# B&R Automation Studio project 305841_E00002_0 (part 10)

#### AxSMInit.st
```iecst
PROGRAM _INIT
  // set ax pointer to the element of the global sMot_Axis array
  ax ACCESS ADR(axes[AXIS_NO]);

  // set the position limits to point to the global permanent variable
  axPositionLimits ACCESS ADR(gr_AxisPositionLimits[AXIS_NO]);

  // Set the axis number and clear the ignore bit
  ax.AxisNo:= AXIS_NO;

  // **** These settings need to be reviewed/set for each axis
  ax.CouplingParameters.SlaveAxisNo := DINT_TO_USINT(AD_UNKNOWN); // No slaves for the CF VFD
  ax.Ignore := FALSE;
  ax.isAxisEndless := TRUE;
  ax.isAxisVirtual := FALSE;
  ax.isAxisInverter := TRUE;

  // Point to the mappMotion axis, and a slave if there is one
  ax.AxisObj := gAxCfPmp; // mappMotion axis -- see mappMotion in cfg view
  ax.SlaveAxisObj := axDummySlave; // slave axis for the handwheel is dynamic

  // Set the restore pos check fb
  // ax.fbCheckRestorePos.Axis := ADR(ax.AxisObj);
  // ax.fbCheckRestorePos.DataAddress := ADR(gr_AxCfVfdRestorePos); // Set this per axis

  // Load the min/max velocity and accel/decel from constants
  ax.MoveParameters.AccelMin := 0.001; // TODO: Not sure of a good value, but it should not be zero.
  ax.MoveParameters.AccelMax := AXIS_CFVFD_MAX_ACCEL;
  ax.MoveParameters.DecelMin := 0.001; // TODO:Not sure of a good value, but it should not be zero.
  ax.MoveParameters.DecelMax:= AXIS_CFVFD_MAX_DECEL;
  ax.MoveParameters.VelocityMin := 0.000;
  ax.MoveParameters.VelocityMax := AXIS_CFVFD_MAX_VELOCITY;

  // **** The settings below don't normally need to be altered

  // set the fb axis references
  ax.fbMpAxisBasic.MpLink := ADR(ax.AxisObj);
  ax.fbReadDrivePos.Axis:= ADR(ax.AxisObj);
  ax.fbGearIn.Master := ADR(ax.AxisObj);
  ax.fbGearIn.Slave := ADR(ax.SlaveAxisObj);
  ax.fbGearOut.Slave := ADR(ax.SlaveAxisObj);
  ax.fbOffsetShift.Slave := ADR(ax.SlaveAxisObj);
  ax.fbPhaseShift.Slave := ADR(ax.SlaveAxisObj);
  ax.fbCamIn.Master := ADR(ax.AxisObj);
  ax.fbCamIn.Slave := ADR(ax.SlaveAxisObj);
  ax.fbCamOut.Slave := ADR(ax.SlaveAxisObj);
  ax.fbUpdateBFbParams._I_Axis := ADR(ax);

  // Set fb reference to local variables
  ax.fbMpAxisBasic.Parameters := ADR(axisBasicParams);

  // Set previous values for motion parameters so changes can be detected
  ax.MoveParametersPrev := ax.MoveParameters;

  // Clear commands and requests
  fctClearMotionCommands(_I_CmdMask := MACM_NOMASK, _IO_Commands := ax.Commands);
  fctClearMotionRequests(_I_ReqMask := MACM_NOMASK, _IO_Commands := ax.Commands);

  // set the move not allowed flag
  ax.Commands.MoveNotAllowed:= TRUE;

  // Set the most primitive status. If the axis is valid, the
  // full status will be updated later once comms is established, and the drive status is updated via MpAxisBasic
  ax.Status.IsCommuncationReady := FALSE;
  ax.Status.IsReadyToPowerOn := FALSE;

END_PROGRAM
```

### Program Logical/PlcLogic/CutProfile/CutProfileCam (IEC) - Calcs and function calls needed to turn the cut profile into a loaded CAM table.

#### CutProfileCam.var - Local variables
```iecst
VAR CONSTANT
  CAM_POINTS : UINT := 250;
END_VAR

VAR

  (* program control *)
  seqCtr : SINT; (* sequence counter *)
  idx : UINT; (* index *)

  (****** Cam related ******)
  (* program control for cam creation *)
  reqCreateCamTable : BOOL := FALSE; (* request to start seq *)
  createCamTableOS : BOOL := FALSE;
  createCamTableDone : BOOL := FALSE;
  camTableId : UINT := 14; (* 1-14, but data type compatible with cam prepare fb *)
  camSeqCtr : SINT; (* sequence counter *)
  camTable : McCamSectionsType; (* local cam sections table *)
  camData : McCamDataType; (* cam data calculated from sections *)
  camPointsMaster : ARRAY[0..CAM_POINTS] OF LREAL;
  camPointsSlave : ARRAY[0..CAM_POINTS] OF LREAL;
  fbCreateCamSections : fbCalcCamSections;
  fbCalcCamFromSections : MC_BR_CalcCamFromSections;
  fbCalcCamPoints : MC_BR_CalcPointsFromCam;
  fbCamPrepare : MC_BR_CamPrepare;
  (* detect changes to cut profile *)
  cutProfileCamLoadedPrev : sWp_CuttingHead; (* previous cut profile loaded into the cam table. *)
  (* BR Str mem fct params *)
  cutProfileBytes : UDINT;
  result : DINT;
  nxtAddr : UDINT;

  (****** Recipe and file related ******)

  (* Local version of the lookup table *)
	depthToAngleLu : sXYTableLu150;

  (* program control for directory creation *)
  reqInitDirs : BOOL := FALSE; (* request to start seq *)
  initDirsOS : BOOL := FALSE;
  initDirsDone : BOOL := FALSE;
  devName : STRING[80]; (* also used for recipe read *)
  dirName : STRING[255];

  (* program control for Depth To Angle Lu recipe registration *)
  pvNameLocalDepthToAngleLu : STRING[100];
  pvNameGloballDepthToAngleLu : STRING[100];
  pvCatagoryDepthToAngleLu : STRING[50];

  (* program control for recipe read/write *)
  recipeReadOverwiteGlobal : BOOL := FALSE;

  recipeReadFileName : STRING[255];
  recipeWriteFileName : STRING[255];

  reqRecipeReadAngleLu : BOOL := FALSE;
  recipeReadAngleLuOS : BOOL := FALSE;
  recipeReadAngleLuDone : BOOL := FALSE;

  reqRecipeWriteAngleLu : BOOL := FALSE;
  recipeWriteAngleLuOS : BOOL := FALSE;
  recipeWriteAngleLuDone : BOOL := FALSE;
  csvHeader : MpRecipeCsvHeaderType;

  (* FileIO fbs *)
  fbDirCreate : DirCreate;

  (* recipe fbs *)
  fbRcpiRegLocalDToALu : MpRecipeRegPar; (* register local Depth To Angle Lu Table to recipe *)
  fbRcpiRegGlobalDToALu : MpRecipeRegPar; (* register global Depth To Angle Lu Table to recipe *)
  fbRecipeCsv : MpRecipeCsv; (* recipe to/from file *)

END_VAR
```

#### CutProfileCam.st - Cyclic code
```iecst
PROGRAM _INIT

  (****** Cam related ******)
  // Set up fb to populate cam sections
  fbCreateCamSections.CamTable := ADR(camTable);
  fbCreateCamSections.DepthToAngle_T1 := ADR(gr_depthToAngleLu.T1);
  fbCreateCamSections.DepthToAngle_T2 := ADR(gr_depthToAngleLu.T2);
  fbCreateCamSections.DepthToAngle_T3 := ADR(gr_depthToAngleLu.T3);
  // Get the length of the cut profile parts of the cutting head configuration
  // This aids in change detection
  cutProfileBytes := ADR(gr_CfgCurrent.cuttingHead.EndOfCutProfile) - ADR(gr_CfgCurrent.cuttingHead.StartOfCutProfile);

  (****** Recipe and file related ******)

  // Setup registration of PV to a recipe
  // Each PV uses a separate registration FB
  // Local Depth To Angle LU Table
  // Use local LU table for recipe access and transfer to/from global when all is well
  pvNameLocalDepthToAngleLu := 'CrCamTbl:depthToAngleLu';
  pvCatagoryDepthToAngleLu := 'DepthToAngle';
  fbRcpiRegLocalDToALu.MpLink := ADR(angleLuRecipeCsv);
  fbRcpiRegLocalDToALu.Enable := FALSE;
  fbRcpiRegLocalDToALu.ErrorReset := FALSE;
  fbRcpiRegLocalDToALu.PVName := ADR(pvNameLocalDepthToAngleLu);
  fbRcpiRegLocalDToALu.Category := ADR(pvCatagoryDepthToAngleLu);
  // set up the fb by calling with enable false, and then set enable
  // true so it is ready to go in cyclic.
  fbRcpiRegLocalDToALu();
  fbRcpiRegLocalDToALu.Enable := TRUE;

  // Global Depth To Angle LU Table
  // Use local LU table for recipe access and transfer to/from global when all is well
  pvNameGloballDepthToAngleLu := 'gr_depthToAngleLu';
  pvCatagoryDepthToAngleLu := 'DepthToAngle';
  fbRcpiRegGlobalDToALu.MpLink := ADR(angleLuRecipeCsv);
  fbRcpiRegGlobalDToALu.Enable := FALSE;
  fbRcpiRegGlobalDToALu.ErrorReset := FALSE;
  fbRcpiRegGlobalDToALu.PVName := ADR(pvNameGloballDepthToAngleLu);
  fbRcpiRegGlobalDToALu.Category := ADR(pvCatagoryDepthToAngleLu);
  // set up the fb by calling with enable false, and then set enable
  // true so it is ready to go in cyclic.
  fbRcpiRegGlobalDToALu();
  fbRcpiRegGlobalDToALu.Enable := TRUE;

  // Set flag to create directories
  reqInitDirs := TRUE; // true will trigger dir setup (creation) after startup
  initDirsOS := FALSE;
  initDirsDone := FALSE;

  // Set flags to control read/write of recipes
  // recipe file names
  recipeReadFileName := 'DepthToAngleLookup_recipe_b.csv';
  recipeWriteFileName := 'DepthToAngleLookup_recipe_b_FromPlc.csv';

  // set whether or not to overwrite the global data on sucessful local read
  recipeReadOverwiteGlobal := FALSE;

  reqRecipeReadAngleLu := FALSE; // set high to read recipe after startup
  recipeReadAngleLuOS := FALSE;
  recipeReadAngleLuDone := FALSE;

  reqRecipeWriteAngleLu := FALSE; // set high to write recipe after startup
  recipeWriteAngleLuOS := FALSE;
  recipeWriteAngleLuDone := FALSE;

 END_PROGRAM

PROGRAM _CYCLIC

  // *****************
  // Cam table: Detect cut profile changes
  // *****************
  // result = brsmemcmp(ADR(Mem1),ADR(Mem2),length), result = 0 when equal
  result := brsmemcmp(ADR(cutProfileCamLoadedPrev.StartOfCutProfile),
                      ADR(gr_CfgCurrent.cuttingHead.StartOfCutProfile),
                      cutProfileBytes);
  // Enable loading the CAM table if it has not been done yet,
  // or if a change is detected, or if the last time there was an error,
  // but the machine cannot be in cycle while a cam table change in made.
  hmiProcessReqs.calCalcTableEnable := (result <> 0 OR NOT createCamTableDone OR camSeqCtr < -1);
  // If a change has been detected, but the table has not been sucessfully loaded, clear the part motion flag
  IF  hmiProcessReqs.calCalcTableEnable AND createCamTableOS THEN
    partMotion.camTableLoaded := FALSE;
  END_IF;

  // *****************
  // Create Cam table on request
  // *****************
  // Set the create cam table request and clear the HMI request upon an HMI request.
  // The logic will handle the rest.
  IF hmiProcessReqs.camReqCalcTable THEN
    reqCreateCamTable := TRUE;
    hmiProcessReqs.camReqCalcTable := FALSE;
  END_IF;

  // On request, calculate and populate cam sections base on cut parameters.
  // Done sucessfully, and camSeqCtr should start from 1, go up, and then end up at -1.
  // Errors result in a more negative camSeqCtr
  // TODO: Deal with errors. Right now the sequence stops, with the camSeqCtr being set to
  // a value more negative than -1.

  IF reqCreateCamTable THEN

    // if the OS is clear, this is the first time thru ...
    // init the seq number and manage flags and OS
    IF NOT createCamTableOS THEN
      // Set the OS so this bit only happens once per req
      createCamTableOS := TRUE;
      // Init the seq ctr
      camSeqCtr := 1;
      // Clear the done flag
      createCamTableDone := FALSE;
      // Clear the hmi request
      hmiProcessReqs.camReqCalcTable := FALSE;
    END_IF;

    IF 1 = camSeqCtr THEN
      // Use cam id 14 for calculated cam table
      camTableId := PROD_CAM_TABLE_ID;
      // Guess the operator will use this cam id
      // TODO: No access to hmiLibraryAxisReqs in OmSaveDev!!

      // Set up to calc the cam sections fb
      // Use the current cutting head configuration for the cut profile

      // Force the finish pass depth to be zero if the option is not chosen
      IF gr_CfgCurrent.cuttingHead.finishingPass THEN
        fbCreateCamSections.FinishPassDepth :=  gr_CfgCurrent.cuttingHead.finishingPassDepth;
      ELSE
        fbCreateCamSections.FinishPassDepth := 0.0;
      END_IF;
      fbCreateCamSections.PassCount := gr_CfgCurrent.cuttingHead.passCount;
      fbCreateCamSections.FinalDepth := gr_CfgCurrent.cuttingHead.totalDepth;
      fbCreateCamSections.CutInAngle := LREAL_TO_REAL(gr_CfgCurrent.cuttingHead.depthAdjAngle);
      fbCreateCamSections.OverCutAngle := LREAL_TO_REAL(gr_CfgCurrent.cuttingHead.cutOverrunAngle);

      // Clear the camTable, camData, and point arrays
      // nxt_adr := brsmemset(ADR(Mem),value,length);
      nxtAddr := brsmemset(ADR(camTable), 0, SIZEOF(camTable));
      nxtAddr := brsmemset(ADR(camData), 0, SIZEOF(camData));
      nxtAddr := brsmemset(ADR(camPointsMaster), 0, SIZEOF(camPointsMaster));
      nxtAddr := brsmemset(ADR(camPointsSlave), 0, SIZEOF(camPointsSlave));

      // Call with enable false to make sure everything is reset and ready to execute with new info
      fbCreateCamSections.Enable := FALSE;
      fbCreateCamSections();
      // onto the next step
      camSeqCtr := 2;
    ELSIF 2 = camSeqCtr THEN
      // Calc the cam sections
      fbCreateCamSections.Enable := TRUE;
      fbCreateCamSections();
      IF fbCreateCamSections.Done AND NOT fbCreateCamSections.Error THEN
        // All done and no error. Move on ...
        // Reset FB and go to next step
        fbCreateCamSections.Enable := FALSE;
        fbCreateCamSections();
        camSeqCtr := 3;
      ELSIF fbCreateCamSections.Done AND fbCreateCamSections.Error THEN
        // Done with an error. Bail out ...
        camSeqCtr := -2;
      END_IF;
    ELSIF 3 = camSeqCtr THEN
      // Set up to calc the cam from the sections
      fbCalcCamFromSections.CamSectionsAddress := ADR(camTable);
      fbCalcCamFromSections.CamDataAddress := ADR(camData);
      // Call with execute false to make sure everything is reset and ready to execute with new info
      fbCalcCamFromSections.Execute := FALSE;
      fbCalcCamFromSections();
      // onto the next step
      camSeqCtr := 4;
    ELSIF 4 = camSeqCtr THEN
      // Calc the cam sections
      fbCalcCamFromSections.Execute := TRUE;
      fbCalcCamFromSections();
      IF fbCalcCamFromSections.Done AND NOT fbCalcCamFromSections.Error THEN
        // All done and no error. Move on ...
        // Reset FB and go to next step
        fbCalcCamFromSections.Execute := FALSE;
        fbCalcCamFromSections();
        camSeqCtr := 5;
      ELSIF NOT fbCalcCamFromSections.Busy AND fbCalcCamFromSections.Error THEN
        // Done with an error. Bail out ...
        camSeqCtr := -4;
      END_IF;
    ELSIF 5 = camSeqCtr THEN
      // Set up to prepare and load the cam data
      fbCamPrepare.Axis := ADR(axes[AD_INNER_ECCENTRIC].AxisObj);
      fbCamPrepare.Cam.DataObjectName := ''; // not used if Cam.DataAdress <> 0
      fbCamPrepare.Cam.DataAdress := ADR(camData); // cam data calculated in fbCalcCamFromSections
      fbCamPrepare.CamID := camTableId;
      // Call with execute false to make sure everything is reset and ready to execute with new info
      fbCamPrepare.Execute := FALSE;
      fbCamPrepare();
      // onto the next step
      camSeqCtr := 6;
    ELSIF 6 = camSeqCtr THEN
      // Prepare and load the cam data
      fbCamPrepare.Execute := TRUE;
      fbCamPrepare();
      IF fbCamPrepare.Done AND NOT fbCamPrepare.Error THEN
        // All done and no error. Move on ...
        // Reset FB and go to next step
        fbCamPrepare.Execute := FALSE;
        fbCamPrepare();
        camSeqCtr := -1;  // TEST: skip fbCalcCamPoints. Getting an error
      ELSIF NOT fbCamPrepare.Busy AND fbCamPrepare.Error THEN
        // Done with an error. Bail out ...
        camSeqCtr := -6;
      END_IF;
    ELSIF 7 = camSeqCtr THEN
      // Set up to calculate cam points
      fbCalcCamPoints.Cam.DataObjectName := ''; // not used if Cam.DataAdress <> 0
      fbCalcCamPoints.Cam.DataAdress := ADR(camData); // cam data calculated in fbCalcCamFromSections
      fbCalcCamPoints.MasterPointsAddress := ADR(camPointsMaster);
      fbCalcCamPoints.SlavePointsAddress := ADR(camPointsSlave);
      fbCalcCamPoints.NumberOfPoints := CAM_POINTS;
      // Call with execute false to make sure everything is reset and ready to execute with new info
      fbCalcCamPoints.Execute := FALSE;
      fbCalcCamPoints();
      // onto the next step
      camSeqCtr := 8;
    ELSIF 8 = camSeqCtr THEN
      // Calcuate points from the cam data
      fbCalcCamPoints.Execute := TRUE;
      fbCalcCamPoints();
      IF fbCalcCamPoints.Done AND NOT fbCalcCamPoints.Error THEN
        // All done and no error. Move on ...
        // reset fb
        fbCalcCamPoints.Execute := FALSE;
        fbCalcCamPoints();
        camSeqCtr := -1;
      ELSIF NOT fbCalcCamPoints.Busy AND fbCalcCamPoints.Error THEN
        // Done with an error. Bail out ...
        camSeqCtr := -8;
      END_IF;
    ELSIF -1 = camSeqCtr THEN
      // All done making cam sections.
      // Getting ready if another request is made.
      // Clear the createCamTable flag and OS and set the done.
      reqCreateCamTable := FALSE;
      createCamTableOS := FALSE; // clear the OS so another initDirs resets things up top
      createCamTableDone := TRUE;
      // Set the flag in part motion
      partMotion.camTableLoaded := TRUE;
      // reset fb
      fbCreateCamSections.Enable := FALSE;
      fbCreateCamSections();
      // Update the previous cut profile values so changes can be detected
      // nxtAddr = brsmemcpy(adr(Dest),adr(Src),length)
      nxtAddr := brsmemcpy(ADR(cutProfileCamLoadedPrev.StartOfCutProfile),
                           ADR(gr_CfgCurrent.cuttingHead.StartOfCutProfile),
                           cutProfileBytes);
    END_IF;
  ELSE
    // createCamTable is false. Clear the OS so we can one time thru it next time
    createCamTableOS := FALSE;
  END_IF;

  // *****************
  // Set up directories
  // *****************
  // Execute FileIO DirCreate async until done or error
  // seqCtr odd: set up DirCreate fb
  // seqCtr even : create dir
  // Use the OS so the directory management can be easily re-run
  // by setting initDirs true (again)
  IF reqInitDirs THEN
    // if the OS is clear, this is the first time thru ...
    // init the seq number and manage flags and OS
    IF NOT initDirsOS THEN
      // Set the OS so this bit only happens once per initDirs
      initDirsOS := TRUE;
      // Init the seq ctr
      seqCtr := 1;
      // Clear the done flag
      initDirsDone := FALSE;
    END_IF;

    IF 1 = seqCtr THEN
      // Setup for first dir
      devName := 'UserPartitionRoot';
      dirName := 'config';
      fbDirCreate.enable := FALSE;
      fbDirCreate.pDevice := ADR(devName);
      fbDirCreate.pName := ADR(dirName);
      fbDirCreate();
      IF ERR_FUB_ENABLE_FALSE = fbDirCreate.status THEN
        seqCtr := 2;
      END_IF;
    ELSIF 2 = seqCtr THEN
      // create first dir
      fbDirCreate.enable := TRUE;
      fbDirCreate();
      IF ERR_OK = fbDirCreate.status OR fiERR_DIR_ALREADY_EXIST = fbDirCreate.status THEN
        // creation okay or not needed
        seqCtr := 3;
      END_IF;
    ELSIF 3 = seqCtr THEN
      // Setup for seconnd dir
      dirName := 'config\recipes';
      // same addresses for device and name
      fbDirCreate.enable := FALSE;
      fbDirCreate();
      IF ERR_FUB_ENABLE_FALSE = fbDirCreate.status THEN
        seqCtr := 4;
      END_IF;
    ELSIF 4 = seqCtr THEN
      // create second dir
      fbDirCreate.enable := TRUE;
      fbDirCreate();
      IF ERR_OK = fbDirCreate.status OR fiERR_DIR_ALREADY_EXIST = fbDirCreate.status THEN
        // creation okay or not needed
        seqCtr := -1;
      END_IF;
    ELSIF -1 = seqCtr THEN
      // All done making directories.
      // Getting ready if another request is made.
      // Clear the initDirs flag and OS and set the done.
     reqInitDirs := FALSE;
     initDirsOS := FALSE; // clear the OS so another initDirs resets things up top
     initDirsDone := TRUE;
     // shut off the fb as a matter of good practice
     fbDirCreate.enable := FALSE;
     fbDirCreate();
    END_IF;
  ELSE
    // initDirs is false. Clear the OS so we can one time thru it next time
    initDirsOS := FALSE;
  END_IF;

  // *****************
  // Read Write Lu Tables to/from recipe
  // *****************

  // Recipe Registration fb should be called all the time, and need to be active
  // when recipe read/write is performed.
  // MpRecipeRegPar was set up in init
  fbRcpiRegLocalDToALu();
  fbRcpiRegGlobalDToALu();

  // **** Read Recipe
  // Treat recipe read as async until done or error
  // seqCtr odd: set up fbRecipeCsv fb
  // seqCtr even : read recipe
  // Use the OS so the read can be easily re-run
  // by setting registerPvs true (again)
  IF NOT reqInitDirs AND initDirsDone AND
      fbRcpiRegLocalDToALu.Active AND NOT fbRcpiRegLocalDToALu.Error AND
      fbRcpiRegGlobalDToALu.Active AND NOT fbRcpiRegGlobalDToALu.Error AND
      reqRecipeReadAngleLu AND NOT reqRecipeWriteAngleLu THEN
    // if the OS is clear, this is the first time thru ...
    // init the seq number and manage flags and OS
    IF NOT recipeReadAngleLuOS THEN
      // Set the OS so this bit only happens once per initDirs
      recipeReadAngleLuOS := TRUE;
      // Set the pv number
      seqCtr := 1;
      // Clear the done flag
      recipeReadAngleLuDone := FALSE;
    END_IF;

    IF 1 = seqCtr THEN
      // Setup for first pv
      devName := 'Recipes';
      pvCatagoryDepthToAngleLu := 'DepthToAngle';
      fbRecipeCsv.MpLink := ADR(angleLuRecipeCsv);
      fbRecipeCsv.Enable := FALSE;
      fbRecipeCsv.ErrorReset := FALSE;
      fbRecipeCsv.DeviceName := ADR(devName);
      fbRecipeCsv.FileName := ADR(recipeReadFileName);
      fbRecipeCsv.Header := ADR(csvHeader);
      fbRecipeCsv.Category := ADR(pvCatagoryDepthToAngleLu);
      fbRecipeCsv.LoadType := mpRECIPE_CSV_LOAD_ALL;
      fbRecipeCsv.Load := TRUE;
      fbRecipeCsv.Save := FALSE;
      fbRecipeCsv.UpdateNotification := FALSE;
      fbRecipeCsv();
      IF NOT fbRecipeCsv.Enable AND NOT fbRecipeCsv.Active AND 0 = fbRecipeCsv.StatusID THEN
        seqCtr := 2;
      END_IF;
    ELSIF 2 = seqCtr THEN
      // read the recipe file and populate the pv
      fbRecipeCsv.Enable := TRUE;
      fbRecipeCsv();
      IF fbRecipeCsv.CommandDone AND NOT fbRecipeCsv.Error THEN
        // read ok
        // If the bit is set, transfer local to the global table -- this global is battery backed retained/permanent
        IF recipeReadOverwiteGlobal THEN
          gr_depthToAngleLu := depthToAngleLu;
          // Now make a version with the X&Y swapped so an depth can be found from an angle
          gr_angleToDepthLu := gr_depthToAngleLu;
          fctSwapTableT3(table := ADR(gr_angleToDepthLu.T1));
          fctSwapTableT3(table := ADR(gr_angleToDepthLu.T2));
          fctSwapTableT3(table := ADR(gr_angleToDepthLu.T3));
        END_IF;
        seqCtr := -1; // all done!
      END_IF;
    ELSIF -1 = seqCtr THEN
      // All done reading the recipe. Deal with flags
      reqRecipeReadAngleLu := FALSE;
      recipeReadAngleLuOS := FALSE; // clear the OS so another registerPv resets things
      recipeReadAngleLuDone := TRUE;
      // shut off the fb as a matter of good practice
      fbRecipeCsv.Enable := FALSE;
      fbRecipeCsv();
    END_IF;
  ELSE
    // Earlier operations not done, or recipeReadAngleLu flag is clear. Clear to OS so we can one time thru it next time
    recipeReadAngleLuOS := FALSE;
  END_IF;

  // **** Write Recipe
  // Treat recipe read as async until done or error
  // seqCtr odd: set up fbRecipeCsv fb
  // seqCtr even : read recipe
  // Use the OS so the read can be easily re-run
  // by setting registerPvs true (again)
  IF NOT reqInitDirs AND initDirsDone AND
      fbRcpiRegLocalDToALu.Active AND NOT fbRcpiRegLocalDToALu.Error AND
      fbRcpiRegGlobalDToALu.Active AND NOT fbRcpiRegGlobalDToALu.Error AND
      reqRecipeWriteAngleLu AND NOT reqRecipeReadAngleLu THEN
    // if the OS is clear, this is the first time thru ...
    // init the seq number and manage flags and OS
    IF NOT recipeWriteAngleLuOS THEN
      // Set the OS so this bit only happens once per initDirs
      recipeWriteAngleLuOS := TRUE;
      // Set the pv number
      seqCtr := 1;
      // Clear the done flag
      recipeWriteAngleLuDone := FALSE;
    END_IF;

    IF 1 = seqCtr THEN
      // Setup for first pv
      devName := 'Recipes';
      pvCatagoryDepthToAngleLu := 'DepthToAngle';
      csvHeader.Name := 'DepthToAngle';
      csvHeader.Description := 'Depths are given in inches, and angles correspond to negative (slave lag) offsets. Source is Robbie Potts Email.';
      csvHeader.Version := 'b';
      csvHeader.DateTime := DT#2022-06-03-14:56;
      fbRecipeCsv.MpLink := ADR(angleLuRecipeCsv);
      fbRecipeCsv.Enable := FALSE;
      fbRecipeCsv.ErrorReset := FALSE;
      fbRecipeCsv.DeviceName := ADR(devName);
      fbRecipeCsv.FileName := ADR(recipeWriteFileName);
      fbRecipeCsv.Header := ADR(csvHeader);
      fbRecipeCsv.Category := ADR(pvCatagoryDepthToAngleLu);
      fbRecipeCsv.LoadType := mpRECIPE_CSV_LOAD_ALL;
      fbRecipeCsv.Load := FALSE;
      fbRecipeCsv.Save := TRUE;
      fbRecipeCsv.UpdateNotification := FALSE;
      fbRecipeCsv();
      IF NOT fbRecipeCsv.Enable AND NOT fbRecipeCsv.Active AND 0 = fbRecipeCsv.StatusID THEN
        seqCtr := 2;
      END_IF;
    ELSIF 2 = seqCtr THEN
      // write pv to recipe file
      fbRecipeCsv.Enable := TRUE;
      fbRecipeCsv();
      IF fbRecipeCsv.CommandDone AND NOT fbRecipeCsv.Error THEN
        // read ok
        seqCtr := -1; // all done!
      END_IF;
    ELSIF -1 = seqCtr THEN
      // All done reading the recipe. Deal with flags
      reqRecipeWriteAngleLu := FALSE;
      recipeWriteAngleLuOS := FALSE; // clear the OS so another registerPv resets things
      recipeWriteAngleLuDone := TRUE;
      // shut off the fb as a matter of good practice
      fbRecipeCsv.Enable := FALSE;
      fbRecipeCsv();
    END_IF;
  ELSE
    // Earlier operations not done, or recipeWriteAngleLu flag is clear. Clear to OS so we can one time thru it next time
    reqRecipeWriteAngleLu := FALSE;
  END_IF;

END_PROGRAM

PROGRAM _EXIT
	(* Insert code here *)

END_PROGRAM
```

#### LocalFunctions.fun
```iecst
FUNCTION_BLOCK fbCalcCamSections (* Calculate the master and slave angles given cut parameters *)
	VAR_INPUT
    Enable : BOOL;
		PassCount : USINT := 1; (* number of passes *)
		FinalDepth : REAL; (* final cut depth, in units of lookup table *)
		FinishPassDepth : REAL := 0.0; (* finishing pass depth. In units of lookup table. Set to 0 for no finish pass. *)
		CutInAngle : REAL; (* degrees *)
		OverCutAngle : REAL; (* degrees *)
		CamTable : REFERENCE TO McCamSectionsType; (* X values master angle, Y values slave angle *)
		DepthToAngle_T1 : REFERENCE TO sXYTableReal50;
		DepthToAngle_T2 : REFERENCE TO sXYTableReal50;
		DepthToAngle_T3 : REFERENCE TO sXYTableReal50;
    PartMotion : REFERENCE TO sPartMotion;
	END_VAR

  VAR_OUTPUT
    Active : BOOL := FALSE;
    Done : BOOL := FALSE;
    Error : BOOL := FALSE;
  END_VAR

	VAR
    _enableOS : BOOL := FALSE;
		_numPasses : USINT; (* conditioned number of passes *)
		_finalDepth : REAL; (* conditioned final cut depth *)
		_finishPassDepth : REAL; (* conditioned finishing pass depth. Set to 0 for no finish pass. *)
		_cutInAngle : REAL; (* conditioned value *)
		_overCutAngle : REAL; (* conditioned value *)
    _seqCtr : SINT; (* sequence counter *)
		_passCtr : USINT; (* pass counter *)
		_incrCutDepth : REAL; (* incremental depth of a nominal pass *)
		_totalPassDepth : REAL; (* accum depth for the pass *)
		_passAngle : REAL;
		_idx : USINT; (* index *)
    (* lookup angle from depth fb *)
    _fbLookupAngle : fbLookUpYValT3;
	END_VAR
END_FUNCTION_BLOCK

FUNCTION fctGetTableNumberT3 : USINT (* Given an X, find which table to look in *)
	VAR_INPUT
		xVal : REAL;
		t1 : REFERENCE TO sXYTableReal50; (* table 1 *)
		t2 : REFERENCE TO sXYTableReal50; (* table 2 *)
		t3 : REFERENCE TO sXYTableReal50; (* table 3 *)
	END_VAR
END_FUNCTION
```

#### LocalFunctions.st
```iecst
// Calculate the master and slave angles given cut parameters
FUNCTION_BLOCK fbCalcCamSections
  IF Enable AND NOT _enableOS THEN
    // Rising edge of enable ... first time thru.

    // set OS
    _enableOS := TRUE;

    // Set active and clear done and error
    Active := TRUE;
    Error := FALSE;
    Done := FALSE;

    // Get setup to lookup an angle given a depth
    // Make sure the lookup tables get loaded in the lookup fb
    // The lookups will come later
    _fbLookupAngle.Enable := FALSE;
    _fbLookupAngle.T1 := ADR(DepthToAngle_T1);
    _fbLookupAngle.T2 := ADR(DepthToAngle_T2);
    _fbLookupAngle.T3 := ADR(DepthToAngle_T3);
    _fbLookupAngle.LoadTables := TRUE;
    _fbLookupAngle();
    _fbLookupAngle.LoadTables := FALSE;

    // **** Condition inputs
    _numPasses := MAX(1, PassCount); // 1 or greater. Otherwise treat as 1
    _finalDepth := ABS(FinalDepth); // must be positive
    _finishPassDepth := MIN(MAX(0.0, FinishPassDepth), _finalDepth); // must be >= 0.0, <= final depth.
    _cutInAngle := ABS(CutInAngle); // must be positive
    _overCutAngle := ABS(OverCutAngle); // must be positive

    // Init the seq counter
    _seqCtr := 1;

  ELSIF Enable AND _enableOS THEN
    // Enable high. Do this stuff over many scans

    IF 1 = _seqCtr THEN
      // **** First step: make the first entry and figure out the incremental cut depth

      // **** First entry in table is 0,0
      // At the beginning of the table, it is assumed the axes are at zero offset (0,0)
      // at the same velocity (which will normally be zero)
      // Specify absolute positions
      CamTable.Section[0].Mode := mcCAMSECTREF_ABSOLUTE;
      CamTable.Section[0].MasterPoint := 0.0;
      CamTable.Section[0].SlavePoint := 0.0;
      // slave to be at a constant velocity
      CamTable.Section[0].FirstDerivative := 1.0; // velocity ratio
      CamTable.Section[0].SecondDerivative := 0.0; // accel ratio
      // next point will be offset. Use polynomial for this -- good general case solution
      CamTable.Section[0].Type := mcCAMSECTLAW_5TH_ORDER_POLYNOM;
      CamTable.Section[0].InflectionPoint := 0.0; // not used for polynomial

      // **** Figure out pass depths and then resulting angles
      // Make cam table entries
      _incrCutDepth := (_finalDepth - _finishPassDepth) / _numPasses; // nominal pass depth
      PartMotion.nominalPassDepth := _incrCutDepth;

      // Ready for the next step
      _passCtr := 1; // Init pass counter. If controlled loop in seq step 2/3.
      _seqCtr := 2;

    ELSIF 2 = _seqCtr OR 3 = _seqCtr THEN
      // **** Second step: Lookup the nominal pass angle
      // **** Third step: Calculate the nominal pass angle

      IF _incrCutDepth > 0.0 THEN
        // normal case where finishing pass < final depth
        // This would be a FOR loop, but I don't want multi-scan async operations
        // to block or cause scan time issues.
        IF _passCtr <= _numPasses THEN
          // depth for this pass
          _totalPassDepth := _incrCutDepth * _passCtr;

          // lookup step
          IF 2 = _seqCtr THEN
            // Look up angle for the needed depth
            _fbLookupAngle(Enable := TRUE, XVal := _totalPassDepth);
            IF _fbLookupAngle.Done AND NOT _fbLookupAngle.Error THEN
              // Lookup was sucessful. Use the looked up value.
              // Force the angle to be positive, as down below the
              // value is subtracted from the master position to force
              // the slave to have a negative offset.
              // Round just for safety so crazy decimal imprecision or rounding does not cause
              // unexpected small differences in cam entries
              _passAngle := fctRound3(_I_src := ABS(_fbLookupAngle.YVal));
              // done with LU fb
              _fbLookupAngle(Enable := FALSE);
              // move to next step
              _seqCtr := 3;
            ELSIF _fbLookupAngle.Done AND _fbLookupAngle.Error THEN
              // Lookup error. Use 0 for the pass angle, and set the error output
              _passAngle := 0.0;
              Error := TRUE;
              // done with LU fb
              _fbLookupAngle(Enable := FALSE);
              // move to next step
              _seqCtr := 3;
            END_IF;

          // calc step (use looked up angle)
          ELSIF 3 = _seqCtr THEN
            // At this point, we have the angle for this pass.
            // This angle is actually the offset angle between the axes.
            // The offset in practice should be negative, meaning the slave lags
            // behind the master by the amount of the offset.
            // Make an entry in the cam table
            // Each pass has an enrty to establish the pass depth,
            // and a second pass to make the cut, which is 1 revolution from the point the
            // depth is established, plus the overcut distance.
            // For a given pass, the first index/position is: ((pass number - 1) * 2) + 1
            // the second index/position is: first index + 1
            // For a given pass, the first master position is: (cutInAngle + pass number) + ((rev + overcut) * (pass number - 1))
            // the second master position is: first position + rev + overcut
            _idx := ((_passCtr - 1) * 2) + 1; // zero based array index position

            // Establish an offset from previous position
            CamTable.Section[_idx].Mode := mcCAMSECTREF_ABSOLUTE;
            CamTable.Section[_idx].MasterPoint := (_cutInAngle * _passCtr) + ((360.0 + _overCutAngle) * (_passCtr - 1));
            CamTable.Section[_idx].SlavePoint := CamTable.Section[idx].MasterPoint - _passAngle;
            // slave to be at a constant velocity
            CamTable.Section[_idx].FirstDerivative := 1.0; // velocity ratio
            CamTable.Section[_idx].SecondDerivative := 0.0; // accel ratio
            // next point will be a stright section.
            CamTable.Section[_idx].Type := mcCAMSECTLAW_STRAIGHT_LINE;
            CamTable.Section[_idx].InflectionPoint := 0.0; // not used for straight line

            // Keep the offset for a revolution + the overcut distance
            CamTable.Section[_idx + 1].Mode := mcCAMSECTREF_ABSOLUTE;
            CamTable.Section[_idx + 1].MasterPoint := CamTable.Section[idx].MasterPoint + (360.0 + _overCutAngle);
            CamTable.Section[_idx + 1].SlavePoint := CamTable.Section[idx + 1].MasterPoint - _passAngle;
            // slave to be at a constant velocity
            CamTable.Section[_idx + 1].FirstDerivative := 1.0; // velocity ratio
            CamTable.Section[_idx + 1].SecondDerivative := 0.0; // accel ratio
            // next point will establish a new offset, so use a polynomial
            CamTable.Section[_idx + 1].Type := mcCAMSECTLAW_5TH_ORDER_POLYNOM;
            CamTable.Section[_idx + 1].InflectionPoint := 0.0; // not used for polynomial

            // Done with calcs for this pass.
            // Set the sequence counter back to 2 so the next angle can be looked up, and
            // increment the pass count.
            _seqCtr := 2;
            _passCtr := _passCtr + 1;
          END_IF; // seq ctr 2 or 3
        ELSE
          // Done with passes. Ready to move on.
          _seqCtr := 4;
        END_IF; // passCtr <= _numPasses
      ELSE // incr cut depth for this pass > 0
        // Special case where finishing pass was entered to be >= final depth.
        // Nothing to do, and this else is here for documentation and as
        // a place holder in case something ends up being needed.
        // The finishing pass is handled next, and will cover this case
        ;
      END_IF // incr cut depth

    ELSIF 4 = _seqCtr OR 5 = _seqCtr THEN
      // **** Forth step: Lookup the nominal pass angle
      // **** Fifth step: Calculate the nominal pass angle

      // If there is a finishing pass, then create cam entries for it

      // After the for loop, passCount will be 1 more than the number of passes.
      // Perfect for the finishing pass, or the retract entry.
      _idx := ((_passCtr - 1) * 2) + 1; // zero based array index position
      IF _finishPassDepth > 0.0 THEN
        // There is a finishing pass
        // By definition, the finishing pass gets us to our final depth,
        // so regardless of the earlier passes, the finishing pass is always
        // at the offset to give the final depth.
        // Look up angle for the needed depth
        IF 4 = _seqCtr THEN
          // Look up angle for the needed depth
          _fbLookupAngle(Enable := TRUE, XVal := _finalDepth);
          IF _fbLookupAngle.Done AND NOT _fbLookupAngle.Error THEN
            // Lookup was sucessful. Use the looked up value.
            // Force the angle to be positive, as down below the
            // value is subtracted from the master position to force
            // the slave to have a negative offset.
            // Round just for safety so crazy decimal imprecision or rounding does not cause
            // unexpected small differences in cam entries
            _passAngle := fctRound3(_I_src := ABS(_fbLookupAngle.YVal));
            // done with LU fb
            _fbLookupAngle(Enable := FALSE);
            // move to next step
            _seqCtr := 5;
          ELSIF _fbLookupAngle.Done AND _fbLookupAngle.Error THEN
            // Lookup error. Use 0 for the pass angle, and set the error output
            _passAngle := 0.0;
            Error := TRUE;
            // done with LU fb
            _fbLookupAngle(Enable := FALSE);
            // move to next step
            _seqCtr := 5;
          END_IF;

        ELSIF 5 = seqCtr THEN
          // Establish an offset from previous position
          CamTable.Section[_idx].Mode := mcCAMSECTREF_ABSOLUTE;
          CamTable.Section[_idx].MasterPoint := (_cutInAngle * _passCtr) + ((360.0 + _overCutAngle) * (_passCtr - 1));
          CamTable.Section[_idx].SlavePoint := CamTable.Section[idx].MasterPoint - _passAngle;
          // slave to be at a constant velocity
          CamTable.Section[_idx].FirstDerivative := 1.0; // velocity ratio
          CamTable.Section[_idx].SecondDerivative := 0.0; // accel ratio
          // next point will be a stright section.
          CamTable.Section[_idx].Type := mcCAMSECTLAW_STRAIGHT_LINE;
          CamTable.Section[_idx].InflectionPoint := 0.0; // not used for straight line

          // Keep the offset for a revolution + the overcut distance
          CamTable.Section[_idx + 1].Mode := mcCAMSECTREF_ABSOLUTE;
          CamTable.Section[_idx + 1].MasterPoint := CamTable.Section[idx].MasterPoint + (360.0 + _overCutAngle);
          CamTable.Section[_idx + 1].SlavePoint := CamTable.Section[idx + 1].MasterPoint - _passAngle;
          // slave to be at a constant velocity
          CamTable.Section[_idx + 1].FirstDerivative := 1.0; // velocity ratio
          CamTable.Section[_idx + 1].SecondDerivative := 0.0; // accel ratio
          // next point will establish a new offset, so use a polynomial
          CamTable.Section[_idx + 1].Type := mcCAMSECTLAW_5TH_ORDER_POLYNOM;
          CamTable.Section[_idx + 1].InflectionPoint := 0.0; // not used for polynomial

          // increment the pass count so similar it can be used for the last entry
          _passCtr := _passCtr + 1;
          // calculate a new index for the last entry, which retracts the cutter
          _idx := ((_passCtr - 1) * 2) + 1; // zero based array index position

          // Done with finishing pass. Ready to move on.
          _seqCtr := 6;
        END_IF; // seq ctr 4 or 5
      ELSE
        // _finishPassDepth = <= 0.0 (no finish pass)
        // Ready to move on
        _seqCtr := 6;
      END_IF; // _finishPassDepth

    // **** Do the last entry to retract the cutting head.
    // passCount will either be number of passes + 1 in the non-finishing pass case,
    // or will be number of passes + 2 in the finishing pass case. idx and passCount
    // were already adjusted in the finishing pass case.

    ELSIF 6 = _seqCtr THEN
      // The last cam entry needs to be of type mcCAMSECTLAW_LAST_POINT
      // Establish a zero offset from previous position
      CamTable.Section[_idx].Mode := mcCAMSECTREF_ABSOLUTE;
      CamTable.Section[_idx].MasterPoint := (_cutInAngle * _passCtr) + ((360.0 + _overCutAngle) * (_passCtr - 1));
      CamTable.Section[_idx].SlavePoint := CamTable.Section[_idx].MasterPoint;
      // slave to be at a constant velocity
      CamTable.Section[_idx].FirstDerivative := 1.0; // velocity ratio
      CamTable.Section[_idx].SecondDerivative := 0.0; // accel ratio
      // next point will be a stright section.
      CamTable.Section[_idx].Type := mcCAMSECTLAW_LAST_POINT;
      CamTable.Section[_idx].InflectionPoint := 0.0; // not used for straight line

      // Since the cam table starts at zero degrees, the total cut distance will be the master point angle at this point
      PartMotion.totalCutDistance := CamTable.Section[_idx].MasterPoint;

      // Done with sequence
      Active := FALSE;
      Done := TRUE;
      _seqCtr := -1;
    END_IF; // seq ctr
  ELSE
    // Not enabled. Clear OS reset outputs.
    _enableOS := FALSE;
    Active := FALSE;
    Done := FALSE;
    Error := FALSE;
  END_IF; // enabled or not

END_FUNCTION_BLOCK

// Given an X, find which of 3 tables to look in
FUNCTION fctGetTableNumberT3
  // Return a 1, 2, or 3 for which table to look in
  // NOTE: X values in each table need to be sorted in ascending order
  // NOTE: It is assumed that x values in table 1 < table 2 < table 3

  // If value is less than or equal the last value in table 1,
  // then the value must represented in or before table 1. Return 1.
  IF xVal <= t1.xVals[t1.numberOfVals - 1] THEN
    fctGetTableNumberT3 := 1;
    RETURN;
  ELSIF xVal >= t3.xVals[0] THEN
    // If value is greater than or equal to the first value in table 3,
    // then the value must be represented in or after table 3. Return 3.
    fctGetTableNumberT3 := 3;
    RETURN;
  ELSE
    // The value must be too big to be represented in table 1,
    // and too small to be represented in table 3.
    // Table 2 is the best choice. Return 2.
    fctGetTableNumberT3 := 2;
    RETURN;
  END_IF;

END_FUNCTION
```

### Program Logical/PlcLogic/CutProfile/PartCfgCalcs (IEC) - Calculate Part motion parameters based on HMI entries.

#### PartCfgCalcs.var - Local variables
```iecst
VAR CONSTANT

END_VAR

VAR
  (* temp values to aid in calculations *)
  calcReal1 : REAL;  (* temporary value *)
  calcLReal1 : LREAL; (* temporary value *)
  calcDint1 : DINT;  (* temporary value *)

  (* detect changes to the machine configuration *)
  wpCfgPrev : sWp_Configuration; (* previous cut profile loaded into the cam table. *)
  (* BR Str mem fct params *)
  wpCfgBytes : UDINT;
  result : DINT;
  nxtAddr : UDINT;

  (* detect changes to the cutting depth *)
  offsetPrev : LREAL := INVALID_SENTINEL_LREAL;

  (* lookup cutter depth from offset angle fb *)
  fbLookupDepth : fbLookUpYValT3;

END_VAR
```

#### PartCfgCalcs.st - Init, cyclic, exit code
```iecst
PROGRAM _INIT
  // Get the length of the configuration
  // This aids in change detection
  wpCfgBytes := ADR(gr_CfgCurrent.startOfCfg) - ADR(gr_CfgCurrent.endOfCfg);

  // Get setup to lookup a depth given an angle
  // Make sure the lookup tables get loaded in the lookup fb
  // The lookups will come later
  fbLookupDepth.Enable := FALSE;
  fbLookupDepth.T1 := ADR(gr_angleToDepthLu.T1);
  fbLookupDepth.T2 := ADR(gr_angleToDepthLu.T2);
  fbLookupDepth.T3 := ADR(gr_angleToDepthLu.T3);
  fbLookupDepth.LoadTables := TRUE;
  fbLookupDepth();
  fbLookupDepth.LoadTables := FALSE;

END_PROGRAM

PROGRAM _CYCLIC
  // *****************
  // Part configuration changes
  // *****************
  //
  // Detect a change
  // result = brsmemcmp(ADR(Mem1),ADR(Mem2),length), result = 0 when equal
  result := brsmemcmp(ADR(wpCfgPrev.startOfCfg),
                      ADR(gr_CfgCurrent.startOfCfg),
                      wpCfgBytes);

  // *****************
  // Depth (eccentric offset angle) changes
  // *****************
  //
  // Detect a change

END_PROGRAM

PROGRAM _EXIT
	(* Insert code here *)

END_PROGRAM
```

#### CalcActions.st
```iecst
ACTION CalcPartMotion :

  // Calc cut velocity
  CalcCutVelocity;

  // Calc pass depth
  CalcPassDepth;

  // Calc depth adjustment velocity.
  // Note this is an average/approximate value for informaitional and approximate use.
  // It does not take into account accel and decel and isn't the exact value the system calculates
  // for coordinated moves.
  CalcDepthAdjVelocity;

  // Calc the number of indexes needed to process a part
  CalcTotalZIndexes;

  // Calc index related values
  CalcZIndex;

END_ACTION

ACTION CalcCutterDepthAct: // Calc cutter depth (mm) from angle
  // Calculated position of the outer eccentric is outer - inner. The lookup table
  // uses positive angles, even though the offset is usualy expressed as being
  // negative, since the inner laggs the outer. Consider it an error if the outer
  // is lagging the inner. The teeth would be at a depth, but now one coverd by the LU table.
  // Allow a small negative offset just so dithering around zero isn't a problem.
  IF axes[AD_OUTER_ECCENTRIC].Status.CalculatedPosition1 <> INVALID_SENTINEL_LREAL AND
      axes[AD_OUTER_ECCENTRIC].Status.CalculatedPosition1 >= -1.0 * ABS(TOL_DEPTH_ZERO_DEG) THEN
    fbLookupDepth(Enable := TRUE, XVal := LREAL_TO_REAL(axes[AD_OUTER_ECCENTRIC].Status.CalculatedPosition1));
    IF fbLookupDepth.Done AND NOT fbLookupDepth.Error THEN
      // Lookup was sucessful. Use the looked up value.
      // Round just for safety so crazy decimal imprecision or rounding does not cause
      // unexpected small differences in cam entries
      partMotion.currentCutterDepth := fctRound3(_I_src := ABS(fbLookupDepth.YVal * 25.4)); // LU in inches, but struct value in in mm
      // done with LU
      fbLookupDepth(Enable := FALSE);
      // Update previous value for change detect
      offsetPrev := axes[AD_OUTER_ECCENTRIC].Status.CalculatedPosition1;

    ELSIF fbLookupDepth.Done AND fbLookupDepth.Error THEN
      // Lookup error. Use invalid for the cutter depth
      partMotion.currentCutterDepth := INVALID_SENTINEL_REAL;
      // done with LU fb
      fbLookupDepth(Enable := FALSE);
      // Update previous value for change detect
      offsetPrev := INVALID_SENTINEL_LREAL;
    END_IF;

END_ACTION

ACTION CalcCutVelocity : // Calc cut velocity in deg/sec from the inside diameter and feed rate
  partMotion.cutVelocity := fctCalcCutVelocity(
  _I_InnerDiameter := gr_PartCurrent.partDfn.nomId,
  _I_FeedRate := gr_CfgCurrent.cuttingHead.feedRate);
END_ACTION

ACTION CalcPassDepth: // Calc pass depth from total depth, number of passes, and finishing pass depth
// Factor in finishing pass
  IF gr_CfgCurrent.cuttingHead.finishingPass THEN
    calcReal1 := MAX(gr_CfgCurrent.cuttingHead.finishingPassDepth, 0.0); // no negative depths
  ELSE
    calcReal1 := 0.0;
  END_IF;

  partMotion.passDepth := fctCalcPassDepth(
  _I_TotalDepth := gr_CfgCurrent.cuttingHead.totalDepth,
  _I_PassCount := gr_CfgCurrent.cuttingHead.passCount,
  _I_FPDepth := calcReal1 ); // calcReal1 at call time has the finishing pass depth
END_ACTION

ACTION CalcTotalZIndexes :
  // Number of indexes to process a part
  // Round up if a partial index is needed
  IF gr_PartCurrent.partDfn.nomCutLength > 0.0 AND gr_CfgCurrent.zAxis.indexDist > 0.0 THEN
    partMotion.totalIndexes := LREAL_TO_USINT(fctLRCeiling(gr_PartCurrent.partDfn.nomCutLength / gr_CfgCurrent.zAxis.indexDist));
  ELSE
    partMotion.totalIndexes := 0;
  END_IF;
END_ACTION

ACTION CalcZIndex :
  // If Z is calibrated, then see where we are for a Z index based on position.
  // Set part current isZIndexed if Z is in an index position.
  // The stat of cut position is subtracted out, and when the head is at
  // the start of cut position, the index should be 1.
  // The general algorithm is index = ((pos - start of cut) / index distance) + 1
  // An
  IF gr_PartCurrent.isZCalibrated THEN
    // Need to know position relative to the start of cut position
    calcLReal1 := axes[AD_Z].Status.Position - gr_CfgCurrent.zAxis.startOfCutPos;
    // Get the Z index count. Value of 0 means the Z position is below the start of cut position, or
    // above the cut length of the workpiece (start of cut pos + cut length, e.g. load/unload position)
    // This is a floating point number that should have a very close to an integer when Z is properly indexed
    IF calcLReal1 < (-1.0 * TOL_ZINDEX) THEN
      // If we are more negative than the tolerance, we are below the start
      // Make the index 0, and call it not indexed
      gr_PartCurrent.zIndexLRCount := 0.0;
      gr_PartCurrent.zIndexCount := 0;
      gr_PartCurrent.isZIndexed := FALSE;
    ELSIF calcLReal1 > (gr_CfgCurrent.zAxis.startOfCutPos + (gr_CfgCurrent.zAxis.indexDist * (partMotion.totalIndexes - 1))) THEN
      // If we are higher than the last index position , we are off the top end.
      // Subtract 1 from totalIndexed, because the Start of Cut is index 1, and there are total indexes - 1 above that.
      // Make the index 0, and call it not indexed
      gr_PartCurrent.zIndexLRCount := 0.0;
      gr_PartCurrent.zIndexCount := 0;
      gr_PartCurrent.isZIndexed := FALSE;
    ELSE
      // If we get here, we are somewhere within the cut length. Consider it indexed if we are at an indexed position.
      gr_PartCurrent.zIndexLRCount := (calcLReal1 / gr_CfgCurrent.zAxis.indexDist) + 1.0;  // Float value for info. SOC is 1, not zero, so we need to add 1
      gr_PartCurrent.zIndexCount := LREAL_TO_USINT(gr_PartCurrent.zIndexLRCount); // Integer index pos, rounded
      // If the position is close enough to an integer index pos, consider us indexed.
      // (Pos - SOC) - the indexed pos from SOC has to be < tolerance
      // TODO: Figure out proper index tolerance. Should correspond to needed Z index precision.
      gr_PartCurrent.isZIndexed := ABS(calcLReal1 - ((gr_PartCurrent.zIndexCount - 1) * gr_CfgCurrent.zAxis.indexDist)) < TOL_ZINDEX;
    END_IF;
  ELSE
    // Not calibrated, so no valid count and not indexed
    gr_PartCurrent.zIndexLRCount := 0.0;
    gr_PartCurrent.zIndexCount := 0;
    gr_PartCurrent.isZIndexed := FALSE;
  END_IF;

END_ACTION

ACTION SetStepTOs :
    gr_ProdModestepTOs[PCS_UNKNOWN]           := T#0ms;
    gr_ProdModestepTOs[PCS_INIT]              := T#0ms;
    gr_ProdModestepTOs[PCS_MODE_CHECK]        := T#0ms;
    gr_ProdModestepTOs[PCS_WAIT_FOR_PROD]     := T#0ms;
    gr_ProdModestepTOs[PCS_WAIT_FOR_START]    := T#0ms;
    gr_ProdModestepTOs[PCS_DECOUPLE_ECC]      := T#0ms;
    gr_ProdModestepTOs[PCS_RESET_AXES]        := T#0ms;
    gr_ProdModestepTOs[PCS_ENABLE_AXES]       := T#0ms;
    gr_ProdModestepTOs[PCS_START_CF]          := T#0ms;
    gr_ProdModestepTOs[PCS_ZERO_DEPTH]        := T#0ms;
    gr_ProdModestepTOs[PCS_Z_TO_SOC]          := T#0ms;
    gr_ProdModestepTOs[PCS_NEXT_CYCLE]        := T#0ms;
    gr_ProdModestepTOs[PCS_START_SPINDLE]     := T#0ms;
    gr_ProdModestepTOs[PCS_COUPLE_ECC]        := T#0ms;
    gr_ProdModestepTOs[PCS_START_PASS]        := T#0ms;
    gr_ProdModestepTOs[PCS_SYNCHING1]         := T#0ms;
    gr_ProdModestepTOs[PCS_SYNCHING2]         := T#0ms;
    gr_ProdModestepTOs[PCS_SYNCHING3]         := T#0ms;
    gr_ProdModestepTOs[PCS_AXES_SYNCHED]      := T#0ms;
    gr_ProdModestepTOs[PCS_SET_NEXT_PASS]     := T#0ms;
    gr_ProdModestepTOs[PCS_SET_FINISH_PASS]   := T#0ms;
    gr_ProdModestepTOs[PCS_SET_RETRACT]       := T#0ms;
    gr_ProdModestepTOs[PCS_STOP_SPINDLE]      := T#0ms;
    gr_ProdModestepTOs[PCS_INDEX_Z_WAIT]      := T#0ms;
    gr_ProdModestepTOs[PCS_CF_OFF1]           := T#0ms;
    gr_ProdModestepTOs[PCS_CF_OFF2]           := T#0ms;
    gr_ProdModestepTOs[PCS_Z_TO_UNLOAD]       := T#0ms;
    gr_ProdModestepTOs[PCS_DONE_WAIT]         := T#0ms;
    gr_ProdModestepTOs[PCS_INDEX_Z]           := T#0ms;
    gr_ProdModestepTOs[PCS_EOC_WAIT]          := T#0ms;
    gr_ProdModestepTOs[PCS_CF_TO]             := T#0ms;
    gr_ProdModestepTOs[PCS_START_CF2]         := T#0ms;
    gr_ProdModestepTOs[PCS_CYCLE_STOP]        := T#0ms;
    gr_ProdModestepTOs[PCS_CS_STOP_AXES]      := T#0ms;
    gr_ProdModestepTOs[PCS_CS_ZERO_DEPTH]     := T#0ms;
    gr_ProdModestepTOs[PCS_CS_STOP_SPINDLE]   := T#0ms;
    gr_ProdModestepTOs[PCS_CS_DISABLE_AXES]   := T#0ms;
    gr_ProdModestepTOs[PCS_CS_STOP_CF]        := T#0ms;

END_ACTION
```

#### LocalFunctions.fun
```iecst
FUNCTION fctCalcPassDepth : REAL (* mm, Return a pass depth base on number of passes and finishing depth *)
  VAR_INPUT
    TotalDepth : REAL; (* mm, final depth *)
    PassCount : USINT; (* number of passes to take, not counting finishing pass *)
    FPDepth : REAL; (* mm, depth of finishing pass. Zero to not have one *)
  END_VAR

  VAR
    _fpDepth : REAL;
  END_VAR
END_FUNCTION

FUNCTION fctCalcCutVelocity : REAL (* deg/sec Return the cut velocity *)
  VAR_INPUT
    InnerDiameter : REAL; (* mm. Inner diameter *)
    FeedRate : REAL; (* mm/sec *)
  END_VAR
END_FUNCTION
```

#### LocalFunctions.st
```iecst
// Return a pass depth based on the number of passes and a finishing depth
FUNCTION fctCalcPassDepth
  // Subtract out the finish pass, and calc the pass depth
  // based on the number of passes, and the total depth.

  // Qualify total depth and pass count. If total depth or pass count
  // is <= 0, then return 0.
  IF TotalDepth <= 0.0 OR PassCount <= 0 THEN
    fctCalcPassDepth := 0.0;
    RETURN;
  END_IF;

  // At this point, total depth and pass count are at least positive values.
  // Qualify finish pass depth -- it can be zero, but it can't be negative or
  // more than the total depth
  _fpDepth := MAX(FPDepth, 0.0);
  _fpDepth := MIN(TotalDepth, _fpDepth);
  fctCalcPassDepth := (TotalDepth - _fpDepth) / USINT_TO_REAL(PassCount);
END_FUNCTION

// Return the cut velocity based on feed rate and inside diameter
FUNCTION fctCalcCutVelocity
  // 360 degrees / circumference * feedrate = feed rate in degrees/sec
  // Do not allow a negative velocity or division by zero or non-sensical inputs. Rtn 0 in these cases.
  IF InnerDiameter <= 0.0 OR FeedRate <= 0.0 THEN
    fctCalcCutVelocity := 0.0;
    RETURN;
  ELSE
    // Inputs are okay. Calc velocity.
    // deg/mm * mm/sec = deg/sec
    fctCalcCutVelocity := (360.0 / (InnerDiameter * brmPI)) * FeedRate;
  END_IF;
END_FUNCTION
```

### Program Logical/PlcLogic/CutProfile/CreateCamTable (IEC)

#### CreateCamTable.st - Cyclic code
```iecst
PROGRAM _INIT

  (****** Cam related ******)
  // Set up fb to populate cam sections
  fbCreateCamSections.CamTable := ADR(camTable);
  fbCreateCamSections.DepthToAngle_T1 := ADR(gr_depthToAngleLu.T1);
  fbCreateCamSections.DepthToAngle_T2 := ADR(gr_depthToAngleLu.T2);
  fbCreateCamSections.DepthToAngle_T3 := ADR(gr_depthToAngleLu.T3);
  // Get the length of the cut profile parts of the cutting head configuration
  // This aids in change detection
  cutProfileBytes := ADR(gr_CfgCurrent.cuttingHead.EndOfCutProfile) - ADR(gr_CfgCurrent.cuttingHead.StartOfCutProfile);

  (****** Recipe and file related ******)
  gr_depthToAngleLu; // Make sure the tables exist!!
  depthToAngleLu;

  // Setup registration of PV to a recipe
  // Each PV uses a separate registration FB
  // Local Depth To Angle LU Table
  // Use local LU table for recipe access and transfer to/from global when all is well
  pvNameLocalDepthToAngleLu := 'CrCamTbl:depthToAngleLu';
  pvCatagoryDepthToAngleLu := 'DepthToAngle';
  fbRcpiRegLocalDToALu.MpLink := ADR(angleLuRecipeCsv);
  fbRcpiRegLocalDToALu.Enable := FALSE;
  fbRcpiRegLocalDToALu.ErrorReset := FALSE;
  fbRcpiRegLocalDToALu.PVName := ADR(pvNameLocalDepthToAngleLu);
  fbRcpiRegLocalDToALu.Category := ADR(pvCatagoryDepthToAngleLu);
  // set up the fb by calling with enable false, and then set enable
  // true so it is ready to go in cyclic.
  fbRcpiRegLocalDToALu();
  fbRcpiRegLocalDToALu.Enable := TRUE;

  // Global Depth To Angle LU Table
  // Use local LU table for recipe access and transfer to/from global when all is well
  pvNameGloballDepthToAngleLu := 'gr_depthToAngleLu';
  pvCatagoryDepthToAngleLu := 'DepthToAngle';
  fbRcpiRegGlobalDToALu.MpLink := ADR(angleLuRecipeCsv);
  fbRcpiRegGlobalDToALu.Enable := FALSE;
  fbRcpiRegGlobalDToALu.ErrorReset := FALSE;
  fbRcpiRegGlobalDToALu.PVName := ADR(pvNameGloballDepthToAngleLu);
  fbRcpiRegGlobalDToALu.Category := ADR(pvCatagoryDepthToAngleLu);
  // set up the fb by calling with enable false, and then set enable
  // true so it is ready to go in cyclic.
  fbRcpiRegGlobalDToALu();
  fbRcpiRegGlobalDToALu.Enable := TRUE;

  // Set flag to create directories
  reqInitDirs := TRUE; // true will trigger dir setup (creation) after startup
  initDirsOS := FALSE;
  initDirsDone := FALSE;

  // Set flags to control read/write of recipes
  // recipe file names
  recipeReadFileName := 'DepthToAngleLookup_recipe_b.csv';
  recipeWriteFileName := 'DepthToAngleLookup_recipe_b_FromPlc.csv';

  // set whether or not to overwrite the global data on sucessful local read
  recipeReadOverwiteGlobal := FALSE;

  reqRecipeReadAngleLu := FALSE; // set high to read recipe after startup
  recipeReadAngleLuOS := FALSE;
  recipeReadAngleLuDone := FALSE;

  reqRecipeWriteAngleLu := FALSE; // set high to write recipe after startup
  recipeWriteAngleLuOS := FALSE;
  recipeWriteAngleLuDone := FALSE;

 END_PROGRAM

PROGRAM _CYCLIC

  // *****************
  // Cam table: Detect cut profile changes
  // *****************
  // result = brsmemcmp(ADR(Mem1),ADR(Mem2),length), result = 0 when equal
  result := brsmemcmp(ADR(cutProfilePrev.StartOfCutProfile),
                      ADR(gr_CfgCurrent.cuttingHead.StartOfCutProfile),
                      cutProfileBytes);
  // Enable loading the CAM table if it has not been done yet,
  // or if a change is detected, or if the last time there was an error,
  // but the machine cannot be in cycle while a cam table change in made.
  hmiProcessReqs.calCalcTableEnable := (result <> 0 OR NOT createCamTableDone OR camSeqCtr < -1);

  // *****************
  // Create Cam table on request
  // *****************
  // Set the create cam table request and clear the HNI request upon an HMI request.
  // The logic will handle the rest.
  IF hmiProcessReqs.camReqCalcTable THEN
    reqCreateCamTable := TRUE;
    hmiProcessReqs.camReqCalcTable := FALSE;
  END_IF;

  // On request, calculate and populate cam sections base on cut parameters.
  // Done sucessfully, and camSeqCtr should start from 1, go up, and then end up at -1.
  // Errors result in a more negative camSeqCtr
  // TODO: Deal with errors. Right now the sequence stops, with the camSeqCtr being set to
  // a value more negative than -1.

  IF reqCreateCamTable THEN

    // if the OS is clear, this is the first time thru ...
    // init the seq number and manage flags and OS
    IF NOT createCamTableOS THEN
      // Set the OS so this bit only happens once per req
      createCamTableOS := TRUE;
      // Init the seq ctr
      camSeqCtr := 1;
      // Clear the done flag
      createCamTableDone := FALSE;
      // Clear the hmi request
      hmiProcessReqs.camReqCalcTable := FALSE;
    END_IF;

    IF 1 = camSeqCtr THEN
      // Use cam id 14 for calculated cam table
      camTableId := PROD_CAM_TABLE_ID;
      // Guess the operator will use this cam id
      // TODO: No access to hmiLibraryAxisReqs in OmSaveDev!!

      // Set up to calc the cam sections fb
      // Use the current cutting head configuration for the cut profile

      // Force the finish pass depth to be zero if the option is not chosen
      IF gr_CfgCurrent.cuttingHead.finishingPass THEN
        fbCreateCamSections.FinishPassDepth :=  gr_CfgCurrent.cuttingHead.finishingPassDepth;
      ELSE
        fbCreateCamSections.FinishPassDepth := 0.0;
      END_IF;
      fbCreateCamSections.PassCount := gr_CfgCurrent.cuttingHead.passCount;
      fbCreateCamSections.FinalDepth := gr_CfgCurrent.cuttingHead.totalDepth;
      fbCreateCamSections.CutInAngle := LREAL_TO_REAL(gr_CfgCurrent.cuttingHead.depthAdjAngle);
      fbCreateCamSections.OverCutAngle := LREAL_TO_REAL(gr_CfgCurrent.cuttingHead.cutOverrunAngle);

      // Clear the camTable, camData, and point arrays
      // nxt_adr := brsmemset(ADR(Mem),value,length);
      nxtAddr := brsmemset(ADR(camTable), 0, SIZEOF(camTable));
      nxtAddr := brsmemset(ADR(camData), 0, SIZEOF(camData));
      nxtAddr := brsmemset(ADR(camPointsMaster), 0, SIZEOF(camPointsMaster));
      nxtAddr := brsmemset(ADR(camPointsSlave), 0, SIZEOF(camPointsSlave));

      // Call with enable false to make sure everything is reset and ready to execute with new info
      fbCreateCamSections.Enable := FALSE;
      fbCreateCamSections();
      // onto the next step
      camSeqCtr := 2;
    ELSIF 2 = camSeqCtr THEN
      // Calc the cam sections
      fbCreateCamSections.Enable := TRUE;
      fbCreateCamSections();
      IF fbCreateCamSections.Done AND NOT fbCreateCamSections.Error THEN
        // All done and no error. Move on ...
        // Reset FB and go to next step
        fbCreateCamSections.Enable := FALSE;
        fbCreateCamSections();
        camSeqCtr := 3;
      ELSIF fbCreateCamSections.Done AND fbCreateCamSections.Error THEN
        // Done with an error. Bail out ...
        camSeqCtr := -2;
      END_IF;
    ELSIF 3 = camSeqCtr THEN
      // Set up to calc the cam from the sections
      fbCalcCamFromSections.CamSectionsAddress := ADR(camTable);
      fbCalcCamFromSections.CamDataAddress := ADR(camData);
      // Call with execute false to make sure everything is reset and ready to execute with new info
      fbCalcCamFromSections.Execute := FALSE;
      fbCalcCamFromSections();
      // onto the next step
      camSeqCtr := 4;
    ELSIF 4 = camSeqCtr THEN
      // Calc the cam sections
      fbCalcCamFromSections.Execute := TRUE;
      fbCalcCamFromSections();
      IF fbCalcCamFromSections.Done AND NOT fbCalcCamFromSections.Error THEN
        // All done and no error. Move on ...
        // Reset FB and go to next step
        fbCalcCamFromSections.Execute := FALSE;
        fbCalcCamFromSections();
        camSeqCtr := 5;
      ELSIF NOT fbCalcCamFromSections.Busy AND fbCalcCamFromSections.Error THEN
        // Done with an error. Bail out ...
        camSeqCtr := -4;
      END_IF;
    ELSIF 5 = camSeqCtr THEN
      // Set up to prepare and load the cam data
      fbCamPrepare.Axis := ADR(axes[AD_INNER_ECCENTRIC].AxisObj);
      fbCamPrepare.Cam.DataObjectName := ''; // not used if Cam.DataAdress <> 0
      fbCamPrepare.Cam.DataAdress := ADR(camData); // cam data calculated in fbCalcCamFromSections
      fbCamPrepare.CamID := camTableId;
      // Call with execute false to make sure everything is reset and ready to execute with new info
      fbCamPrepare.Execute := FALSE;
      fbCamPrepare();
      // onto the next step
      camSeqCtr := 6;
    ELSIF 6 = camSeqCtr THEN
      // Prepare and load the cam data
      fbCamPrepare.Execute := TRUE;
      fbCamPrepare();
      IF fbCamPrepare.Done AND NOT fbCamPrepare.Error THEN
        // All done and no error. Move on ...
        // Reset FB and go to next step
        fbCamPrepare.Execute := FALSE;
        fbCamPrepare();
        camSeqCtr := -1;  // TEST: skip fbCalcCamPoints. Getting an error
      ELSIF NOT fbCamPrepare.Busy AND fbCamPrepare.Error THEN
        // Done with an error. Bail out ...
        camSeqCtr := -6;
      END_IF;
    ELSIF 7 = camSeqCtr THEN
      // Set up to calculate cam points
      fbCalcCamPoints.Cam.DataObjectName := ''; // not used if Cam.DataAdress <> 0
      fbCalcCamPoints.Cam.DataAdress := ADR(camData); // cam data calculated in fbCalcCamFromSections
      fbCalcCamPoints.MasterPointsAddress := ADR(camPointsMaster);
      fbCalcCamPoints.SlavePointsAddress := ADR(camPointsSlave);
      fbCalcCamPoints.NumberOfPoints := CAM_POINTS;
      // Call with execute false to make sure everything is reset and ready to execute with new info
      fbCalcCamPoints.Execute := FALSE;
      fbCalcCamPoints();
      // onto the next step
      camSeqCtr := 8;
    ELSIF 8 = camSeqCtr THEN
      // Calcuate points from the cam data
      fbCalcCamPoints.Execute := TRUE;
      fbCalcCamPoints();
      IF fbCalcCamPoints.Done AND NOT fbCalcCamPoints.Error THEN
        // All done and no error. Move on ...
        // reset fb
        fbCalcCamPoints.Execute := FALSE;
        fbCalcCamPoints();
        camSeqCtr := -1;
      ELSIF NOT fbCalcCamPoints.Busy AND fbCalcCamPoints.Error THEN
        // Done with an error. Bail out ...
        camSeqCtr := -8;
      END_IF;
    ELSIF -1 = camSeqCtr THEN
      // All done making cam sections.
      // Getting ready if another request is made.
      // Clear the createCamTable flag and OS and set the done.
      reqCreateCamTable := FALSE;
      createCamTableOS := FALSE; // clear the OS so another initDirs resets things up top
      createCamTableDone := TRUE;
      // reset fb
      fbCreateCamSections.Enable := FALSE;
      fbCreateCamSections();
      // Update the previous cut profile values so changes can be detected
      // nxtAddr = brsmemcpy(adr(Dest),adr(Src),length)
      nxtAddr := brsmemcpy(ADR(cutProfilePrev.StartOfCutProfile),
                           ADR(gr_CfgCurrent.cuttingHead.StartOfCutProfile),
                           cutProfileBytes);
    END_IF;
  ELSE
    // createCamTable is false. Clear the OS so we can one time thru it next time
    createCamTableOS := FALSE;
  END_IF;

  // *****************
  // Set up directories
  // *****************
  // Execute FileIO DirCreate async until done or error
  // seqCtr odd: set up DirCreate fb
  // seqCtr even : create dir
  // Use the OS so the directory management can be easily re-run
  // by setting initDirs true (again)
  IF reqInitDirs THEN
    // if the OS is clear, this is the first time thru ...
    // init the seq number and manage flags and OS
    IF NOT initDirsOS THEN
      // Set the OS so this bit only happens once per initDirs
      initDirsOS := TRUE;
      // Init the seq ctr
      seqCtr := 1;
      // Clear the done flag
      initDirsDone := FALSE;
    END_IF;

    IF 1 = seqCtr THEN
      // Setup for first dir
      devName := 'UserPartitionRoot';
      dirName := 'config';
      fbDirCreate.enable := FALSE;
      fbDirCreate.pDevice := ADR(devName);
      fbDirCreate.pName := ADR(dirName);
      fbDirCreate();
      IF ERR_FUB_ENABLE_FALSE = fbDirCreate.status THEN
        seqCtr := 2;
      END_IF;
    ELSIF 2 = seqCtr THEN
      // create first dir
      fbDirCreate.enable := TRUE;
      fbDirCreate();
      IF ERR_OK = fbDirCreate.status OR fiERR_DIR_ALREADY_EXIST = fbDirCreate.status THEN
        // creation okay or not needed
        seqCtr := 3;
      END_IF;
    ELSIF 3 = seqCtr THEN
      // Setup for seconnd dir
      dirName := 'config\recipes';
      // same addresses for device and name
      fbDirCreate.enable := FALSE;
      fbDirCreate();
      IF ERR_FUB_ENABLE_FALSE = fbDirCreate.status THEN
        seqCtr := 4;
      END_IF;
    ELSIF 4 = seqCtr THEN
      // create second dir
      fbDirCreate.enable := TRUE;
      fbDirCreate();
      IF ERR_OK = fbDirCreate.status OR fiERR_DIR_ALREADY_EXIST = fbDirCreate.status THEN
        // creation okay or not needed
        seqCtr := -1;
      END_IF;
    ELSIF -1 = seqCtr THEN
      // All done making directories.
      // Getting ready if another request is made.
      // Clear the initDirs flag and OS and set the done.
     reqInitDirs := FALSE;
     initDirsOS := FALSE; // clear the OS so another initDirs resets things up top
     initDirsDone := TRUE;
     // shut off the fb as a matter of good practice
     fbDirCreate.enable := FALSE;
     fbDirCreate();
    END_IF;
  ELSE
    // initDirs is false. Clear the OS so we can one time thru it next time
    initDirsOS := FALSE;
  END_IF;

  // *****************
  // Read Write Lu Tables to/from recipe
  // *****************

  // Recipe Registration fb should be called all the time, and need to be active
  // when recipe read/write is performed.
  // MpRecipeRegPar was set up in init
  fbRcpiRegLocalDToALu();
  fbRcpiRegGlobalDToALu();

  // **** Read Recipe
  // Treat recipe read as async until done or error
  // seqCtr odd: set up fbRecipeCsv fb
  // seqCtr even : read recipe
  // Use the OS so the read can be easily re-run
  // by setting registerPvs true (again)
  IF NOT reqInitDirs AND initDirsDone AND
      fbRcpiRegLocalDToALu.Active AND NOT fbRcpiRegLocalDToALu.Error AND
      fbRcpiRegGlobalDToALu.Active AND NOT fbRcpiRegGlobalDToALu.Error AND
      reqRecipeReadAngleLu AND NOT reqRecipeWriteAngleLu THEN
    // if the OS is clear, this is the first time thru ...
    // init the seq number and manage flags and OS
    IF NOT recipeReadAngleLuOS THEN
      // Set the OS so this bit only happens once per initDirs
      recipeReadAngleLuOS := TRUE;
      // Set the pv number
      seqCtr := 1;
      // Clear the done flag
      recipeReadAngleLuDone := FALSE;
    END_IF;

    IF 1 = seqCtr THEN
      // Setup for first pv
      devName := 'Recipes';
      pvCatagoryDepthToAngleLu := 'DepthToAngle';
      fbRecipeCsv.MpLink := ADR(angleLuRecipeCsv);
      fbRecipeCsv.Enable := FALSE;
      fbRecipeCsv.ErrorReset := FALSE;
      fbRecipeCsv.DeviceName := ADR(devName);
      fbRecipeCsv.FileName := ADR(recipeReadFileName);
      fbRecipeCsv.Header := ADR(csvHeader);
      fbRecipeCsv.Category := ADR(pvCatagoryDepthToAngleLu);
      fbRecipeCsv.LoadType := mpRECIPE_CSV_LOAD_ALL;
      fbRecipeCsv.Load := TRUE;
      fbRecipeCsv.Save := FALSE;
      fbRecipeCsv.UpdateNotification := FALSE;
      fbRecipeCsv();
      IF NOT fbRecipeCsv.Enable AND NOT fbRecipeCsv.Active AND 0 = fbRecipeCsv.StatusID THEN
        seqCtr := 2;
      END_IF;
    ELSIF 2 = seqCtr THEN
      // read the recipe file and populate the pv
      fbRecipeCsv.Enable := TRUE;
      fbRecipeCsv();
      IF fbRecipeCsv.CommandDone AND NOT fbRecipeCsv.Error THEN
        // read ok
        // If the bit is set, transfer local to the global table -- thisglobal is battery backed retained/permanent
        IF recipeReadOverwiteGlobal THEN
          gr_depthToAngleLu := depthToAngleLu;
        END_IF;
        seqCtr := -1; // all done!
      END_IF;
    ELSIF -1 = seqCtr THEN
      // All done reading the recipe. Deal with flags
      reqRecipeReadAngleLu := FALSE;
      recipeReadAngleLuOS := FALSE; // clear the OS so another registerPv resets things
      recipeReadAngleLuDone := TRUE;
      // shut off the fb as a matter of good practice
      fbRecipeCsv.Enable := FALSE;
      fbRecipeCsv();
    END_IF;
  ELSE
    // Earlier operations not done, or recipeReadAngleLu flag is clear. Clear to OS so we can one time thru it next time
    recipeReadAngleLuOS := FALSE;
  END_IF;

  // **** Write Recipe
  // Treat recipe read as async until done or error
  // seqCtr odd: set up fbRecipeCsv fb
  // seqCtr even : read recipe
  // Use the OS so the read can be easily re-run
  // by setting registerPvs true (again)
  IF NOT reqInitDirs AND initDirsDone AND
      fbRcpiRegLocalDToALu.Active AND NOT fbRcpiRegLocalDToALu.Error AND
      fbRcpiRegGlobalDToALu.Active AND NOT fbRcpiRegGlobalDToALu.Error AND
      reqRecipeWriteAngleLu AND NOT reqRecipeReadAngleLu THEN
    // if the OS is clear, this is the first time thru ...
    // init the seq number and manage flags and OS
    IF NOT recipeWriteAngleLuOS THEN
      // Set the OS so this bit only happens once per initDirs
      recipeWriteAngleLuOS := TRUE;
      // Set the pv number
      seqCtr := 1;
      // Clear the done flag
      recipeWriteAngleLuDone := FALSE;
    END_IF;

    IF 1 = seqCtr THEN
      // Setup for first pv
      devName := 'Recipes';
      pvCatagoryDepthToAngleLu := 'DepthToAngle';
      csvHeader.Name := 'DepthToAngle';
      csvHeader.Description := 'Depths are given in inches, and angles correspond to negative (slave lag) offsets. Source is Robbie Potts Email.';
      csvHeader.Version := 'b';
      csvHeader.DateTime := DT#2022-06-03-14:56;
      fbRecipeCsv.MpLink := ADR(angleLuRecipeCsv);
      fbRecipeCsv.Enable := FALSE;
      fbRecipeCsv.ErrorReset := FALSE;
      fbRecipeCsv.DeviceName := ADR(devName);
      fbRecipeCsv.FileName := ADR(recipeWriteFileName);
      fbRecipeCsv.Header := ADR(csvHeader);
      fbRecipeCsv.Category := ADR(pvCatagoryDepthToAngleLu);
      fbRecipeCsv.LoadType := mpRECIPE_CSV_LOAD_ALL;
      fbRecipeCsv.Load := FALSE;
      fbRecipeCsv.Save := TRUE;
      fbRecipeCsv.UpdateNotification := FALSE;
      fbRecipeCsv();
      IF NOT fbRecipeCsv.Enable AND NOT fbRecipeCsv.Active AND 0 = fbRecipeCsv.StatusID THEN
        seqCtr := 2;
      END_IF;
    ELSIF 2 = seqCtr THEN
      // write pv to recipe file
      fbRecipeCsv.Enable := TRUE;
      fbRecipeCsv();
      IF fbRecipeCsv.CommandDone AND NOT fbRecipeCsv.Error THEN
        // read ok
        seqCtr := -1; // all done!
      END_IF;
    ELSIF -1 = seqCtr THEN
      // All done reading the recipe. Deal with flags
      reqRecipeWriteAngleLu := FALSE;
      recipeWriteAngleLuOS := FALSE; // clear the OS so another registerPv resets things
      recipeWriteAngleLuDone := TRUE;
      // shut off the fb as a matter of good practice
      fbRecipeCsv.Enable := FALSE;
      fbRecipeCsv();
    END_IF;
  ELSE
    // Earlier operations not done, or recipeWriteAngleLu flag is clear. Clear to OS so we can one time thru it next time
    reqRecipeWriteAngleLu := FALSE;
  END_IF;

END_PROGRAM

PROGRAM _EXIT
	(* Insert code here *)

END_PROGRAM
```

#### LocalFunctions.fun
```iecst
FUNCTION_BLOCK fbCalcCamSections (* Calculate the master and slave angles given cut parameters *)
	VAR_INPUT
    Enable : BOOL;
		PassCount : USINT := 1; (* number of passes *)
		FinalDepth : REAL; (* final cut depth, in units of lookup table *)
		FinishPassDepth : REAL := 0.0; (* finishing pass depth. In units of lookup table. Set to 0 for no finish pass. *)
		CutInAngle : REAL; (* degrees *)
		OverCutAngle : REAL; (* degrees *)
		CamTable : REFERENCE TO McCamSectionsType; (* X values master angle, Y values slave angle *)
		DepthToAngle_T1 : REFERENCE TO sXYTableReal50;
		DepthToAngle_T2 : REFERENCE TO sXYTableReal50;
		DepthToAngle_T3 : REFERENCE TO sXYTableReal50;
	END_VAR

  VAR_OUTPUT
    Active : BOOL := FALSE;
    Done : BOOL := FALSE;
    Error : BOOL := FALSE;
  END_VAR

	VAR
    enableOS : BOOL := FALSE;
		_numPasses : USINT; (* conditioned number of passes *)
		_finalDepth : REAL; (* conditioned final cut depth *)
		_finishPassDepth : REAL; (* conditioned finishing pass depth. Set to 0 for no finish pass. *)
		_cutInAngle : REAL; (* conditioned value *)
		_overCutAngle : REAL; (* conditioned value *)
    seqCtr : SINT; (* sequence counter *)
		passCtr : USINT; (* pass counter *)
		incrCutDepth : REAL; (* incremental depth of a nominal pass *)
		totalPassDepth : REAL; (* accum depth for the pass *)
		passAngle : REAL;
		idx : USINT; (* index *)
    (* lookup angle from depth fb *)
    fbLookupAngle : fbLookUpYValT3;
	END_VAR
END_FUNCTION_BLOCK

FUNCTION fctGetTableNumberT3 : USINT (* Given an X, find which table to look in *)
	VAR_INPUT
		xVal : REAL;
		t1 : REFERENCE TO sXYTableReal50; (* table 1 *)
		t2 : REFERENCE TO sXYTableReal50; (* table 2 *)
		t3 : REFERENCE TO sXYTableReal50; (* table 3 *)
	END_VAR
END_FUNCTION

FUNCTION fctSwapTableT3 : USINT (* Swap X & Y columns *)
	VAR_INPUT
		table : REFERENCE TO sXYTableReal50; (* table to swap the X & Y values of *)
	END_VAR
	VAR
		tVals : ARRAY[0..49] OF REAL; (* temporary storage *)
		length : UDINT; (* mem copy length in bytes *)
		nextAddr : UDINT; (* return from memcpy *)
	END_VAR
END_FUNCTION
```

#### LocalFunctions.st
```iecst
// Calculate the master and slave angles given cut parameters
FUNCTION_BLOCK fbCalcCamSections
  IF Enable AND NOT enableOS THEN
    // Rising edge of enable ... first time thru.

    // set OS
    enableOS := TRUE;

    // Set active and clear done and error
    Active := TRUE;
    Error := FALSE;
    Done := FALSE;

    // Make sure the lookup tables get loaded in the lookup fb
    // The lookups will come later
    fbLookupAngle.Enable := FALSE;
    fbLookupAngle.T1 := ADR(DepthToAngle_T1);
    fbLookupAngle.T2 := ADR(DepthToAngle_T2);
    fbLookupAngle.T3 := ADR(DepthToAngle_T3);
    fbLookupAngle.LoadTables := TRUE;
    fbLookupAngle();
    fbLookupAngle.LoadTables := FALSE;

    // **** Condition inputs
    _numPasses := MAX(1, PassCount); // 1 or greater. Otherwise treat as 1
    _finalDepth := ABS(FinalDepth); // must be positive
    _finishPassDepth := MIN(MAX(0.0, FinishPassDepth), _finalDepth); // must be >= 0.0, <= final depth.
    _cutInAngle := ABS(CutInAngle); // must be positive
    _overCutAngle := ABS(OverCutAngle); // must be positive

    // Init the seq counter
    seqCtr := 1;

  ELSIF Enable AND enableOS THEN
    // Enable high. Do this stuff over many scans

    IF 1 = seqCtr THEN
      // **** First step: make the first entry and figure out the incremental cut depth

      // **** First entry in table is 0,0
      // At the beginning of the table, it is assumed the axes are at zero offset (0,0)
      // at the same velocity (which will normally be zero)
      // Specify absolute positions
      CamTable.Section[0].Mode := mcCAMSECTREF_ABSOLUTE;
      CamTable.Section[0].MasterPoint := 0.0;
      CamTable.Section[0].SlavePoint := 0.0;
      // slave to be at a constant velocity
      CamTable.Section[0].FirstDerivative := 1.0; // velocity ratio
      CamTable.Section[0].SecondDerivative := 0.0; // accel ratio
      // next point will be offset. Use polynomial for this -- good general case solution
      CamTable.Section[0].Type := mcCAMSECTLAW_5TH_ORDER_POLYNOM;
      CamTable.Section[0].InflectionPoint := 0.0; // not used for polynomial

      // **** Figure out pass depths and then resulting angles
      // Make cam table entries
      incrCutDepth := (_finalDepth - _finishPassDepth) / _numPasses;

      // Ready for the next step
      passCtr := 1; // Init pass counter. If controlled loop in seq step 2/3.
      seqCtr := 2;

    ELSIF 2 = seqCtr OR 3 = seqCtr THEN
      // **** Second step: Lookup the nominal pass angle
      // **** Third step: Calculate the nominal pass angle

      IF incrCutDepth > 0.0 THEN
        // normal case where finishing pass < final depth
        // This would be a FOR loop, but I don't want multi-scan async operations
        // to block or cause scan time issues.
        IF passCtr <= _numPasses THEN
          // depth for this pass
          totalPassDepth := incrCutDepth * passCtr;

          // lookup step
          IF 2 = seqCtr THEN
            // Look up angle for the needed depth
            fbLookupAngle(Enable := TRUE, XVal := totalPassDepth);
            IF fbLookupAngle.Done AND NOT fbLookupAngle.Error THEN
              // Lookup was sucessful. Use the looked up value.
              // Force the angle to be positive, as down below the
              // value is subtracted from the master position to force
              // the slave to have a negative offset.
              // Round just for safety so crazy decimal imprecision or rounding does not cause
              // unexpected small differences in cam entries
              passAngle := fctRound3(_I_src := ABS(fbLookupAngle.YVal));
              // done with LU fb
              fbLookupAngle(Enable := FALSE);
              // move to next step
              seqCtr := 3;
            ELSIF fbLookupAngle.Done AND fbLookupAngle.Error THEN
              // Lookup error. Use 0 for the pass angle, and set the error output
              passAngle := 0.0;
              Error := TRUE;
              // done with LU fb
              fbLookupAngle(Enable := FALSE);
              // move to next step
              seqCtr := 3;
            END_IF;

          // calc step (use looked up angle)
          ELSIF 3 = seqCtr THEN
            // At this point, we have the angle for this pass.
            // This angle is actually the offset angle between the axes.
            // The offset in practice should be negative, meaning the slave lags
            // behind the master by the amount of the offset.
            // Make an entry in the cam table
            // Each pass has an enrty to establish the pass depth,
            // and a second pass to make the cut, which is 1 revolution from the point the
            // depth is established, plus the overcut distance.
            // For a given pass, the first index/position is: ((pass number - 1) * 2) + 1
            // the second index/position is: first index + 1
            // For a given pass, the first master position is: (cutInAngle + pass number) + ((rev + overcut) * (pass number - 1))
            // the second master position is: first position + rev + overcut
            idx := ((passCtr - 1) * 2) + 1; // zero based array index position

            // Establish an offset from previous position
            CamTable.Section[idx].Mode := mcCAMSECTREF_ABSOLUTE;
            CamTable.Section[idx].MasterPoint := (_cutInAngle * passCtr) + ((360.0 + _overCutAngle) * (passCtr - 1));
            CamTable.Section[idx].SlavePoint := CamTable.Section[idx].MasterPoint - passAngle;
            // slave to be at a constant velocity
            CamTable.Section[idx].FirstDerivative := 1.0; // velocity ratio
            CamTable.Section[idx].SecondDerivative := 0.0; // accel ratio
            // next point will be a stright section.
            CamTable.Section[idx].Type := mcCAMSECTLAW_STRAIGHT_LINE;
            CamTable.Section[idx].InflectionPoint := 0.0; // not used for straight line

            // Keep the offset for a revolution + the overcut distance
            CamTable.Section[idx + 1].Mode := mcCAMSECTREF_ABSOLUTE;
            CamTable.Section[idx + 1].MasterPoint := CamTable.Section[idx].MasterPoint + (360.0 + _overCutAngle);
            CamTable.Section[idx + 1].SlavePoint := CamTable.Section[idx + 1].MasterPoint - passAngle;
            // slave to be at a constant velocity
            CamTable.Section[idx + 1].FirstDerivative := 1.0; // velocity ratio
            CamTable.Section[idx + 1].SecondDerivative := 0.0; // accel ratio
            // next point will establish a new offset, so use a polynomial
            CamTable.Section[idx + 1].Type := mcCAMSECTLAW_5TH_ORDER_POLYNOM;
            CamTable.Section[idx + 1].InflectionPoint := 0.0; // not used for polynomial

            // Done with calcs for this pass.
            // Set the sequence counter back to 2 so the next angle can be looked up, and
            // increment the pass count.
            seqCtr := 2;
            passCtr := passCtr + 1;
          END_IF; // seq ctr 2 or 3
        ELSE
          // Done with passes. Ready to move on.
          seqCtr := 4;
        END_IF; // passCtr <= _numPasses
      ELSE // incr cut depth for this pass > 0
        // Special case where finishing pass was entered to be >= final depth.
        // Nothing to do, and this else is here for documentation and as
        // a place holder in case something ends up being needed.
        // The finishing pass is handled next, and will cover this case
        ;
      END_IF // incr cut depth

    ELSIF 4 = seqCtr OR 5 = seqCtr THEN
      // **** Forth step: Lookup the nominal pass angle
      // **** Fifth step: Calculate the nominal pass angle

      // If there is a finishing pass, then create cam entries for it

      // After the for loop, passCount will be 1 more than the number of passes.
      // Perfect for the finishing pass, or the retract entry.
      idx := ((passCtr - 1) * 2) + 1; // zero based array index position
      IF _finishPassDepth > 0.0 THEN
        // There is a finishing pass
        // By definition, the finishing pass gets us to our final depth,
        // so regardless of the earlier passes, the finishing pass is always
        // at the offset to give the final depth.
        // Look up angle for the needed depth
        IF 4 = seqCtr THEN
          // Look up angle for the needed depth
          fbLookupAngle(Enable := TRUE, XVal := _finalDepth);
          IF fbLookupAngle.Done AND NOT fbLookupAngle.Error THEN
            // Lookup was sucessful. Use the looked up value.
            // Force the angle to be positive, as down below the
            // value is subtracted from the master position to force
            // the slave to have a negative offset.
            // Round just for safety so crazy decimal imprecision or rounding does not cause
            // unexpected small differences in cam entries
            passAngle := fctRound3(_I_src := ABS(fbLookupAngle.YVal));
            // done with LU fb
            fbLookupAngle(Enable := FALSE);
            // move to next step
            seqCtr := 5;
          ELSIF fbLookupAngle.Done AND fbLookupAngle.Error THEN
            // Lookup error. Use 0 for the pass angle, and set the error output
            passAngle := 0.0;
            Error := TRUE;
            // done with LU fb
            fbLookupAngle(Enable := FALSE);
            // move to next step
            seqCtr := 5;
          END_IF;

        ELSIF 5 = seqCtr THEN
          // Establish an offset from previous position
          CamTable.Section[idx].Mode := mcCAMSECTREF_ABSOLUTE;
          CamTable.Section[idx].MasterPoint := (_cutInAngle * passCtr) + ((360.0 + _overCutAngle) * (passCtr - 1));
          CamTable.Section[idx].SlavePoint := CamTable.Section[idx].MasterPoint - passAngle;
          // slave to be at a constant velocity
          CamTable.Section[idx].FirstDerivative := 1.0; // velocity ratio
          CamTable.Section[idx].SecondDerivative := 0.0; // accel ratio
          // next point will be a stright section.
          CamTable.Section[idx].Type := mcCAMSECTLAW_STRAIGHT_LINE;
          CamTable.Section[idx].InflectionPoint := 0.0; // not used for straight line

          // Keep the offset for a revolution + the overcut distance
          CamTable.Section[idx + 1].Mode := mcCAMSECTREF_ABSOLUTE;
          CamTable.Section[idx + 1].MasterPoint := CamTable.Section[idx].MasterPoint + (360.0 + _overCutAngle);
          CamTable.Section[idx + 1].SlavePoint := CamTable.Section[idx + 1].MasterPoint - passAngle;
          // slave to be at a constant velocity
          CamTable.Section[idx + 1].FirstDerivative := 1.0; // velocity ratio
          CamTable.Section[idx + 1].SecondDerivative := 0.0; // accel ratio
          // next point will establish a new offset, so use a polynomial
          CamTable.Section[idx + 1].Type := mcCAMSECTLAW_5TH_ORDER_POLYNOM;
          CamTable.Section[idx + 1].InflectionPoint := 0.0; // not used for polynomial

          // increment the pass count so similar it can be used for the last entry
          passCtr := passCtr + 1;
          // calculate a new index for the last entry, which retracts the cutter
          idx := ((passCtr - 1) * 2) + 1; // zero based array index position

          // Done with finishing pass. Ready to move on.
          seqCtr := 6;
        END_IF; // seq ctr 4 or 5
      ELSE
        // _finishPassDepth = <= 0.0 (no finish pass)
        // Ready to move on
        seqCtr := 6;
      END_IF; // _finishPassDepth

    // **** Do the last entry to retract the cutting head.
    // passCount will either be number of passes + 1 in the non-finishing pass case,
    // or will be number of passes + 2 in the finishing pass case. idx and passCount
    // were already adjusted in the finishing pass case.

    ELSIF 6 = seqCtr THEN
      // The last cam entry needs to be of type mcCAMSECTLAW_LAST_POINT
      // Establish a zero offset from previous position
      CamTable.Section[idx].Mode := mcCAMSECTREF_ABSOLUTE;
      CamTable.Section[idx].MasterPoint := (_cutInAngle * passCtr) + ((360.0 + _overCutAngle) * (passCtr - 1));
      CamTable.Section[idx].SlavePoint := CamTable.Section[idx].MasterPoint;
      // slave to be at a constant velocity
      CamTable.Section[idx].FirstDerivative := 1.0; // velocity ratio
      CamTable.Section[idx].SecondDerivative := 0.0; // accel ratio
      // next point will be a stright section.
      CamTable.Section[idx].Type := mcCAMSECTLAW_LAST_POINT;
      CamTable.Section[idx].InflectionPoint := 0.0; // not used for straight line

      // Done with sequence
      Active := FALSE;
      Done := TRUE;
      seqCtr := -1;
    END_IF; // seq ctr
  ELSE
    // Not enabled. Clear OS reset outputs.
    enableOS := FALSE;
    Active := FALSE;
    Done := FALSE;
    Error := FALSE;
  END_IF; // enabled or not

END_FUNCTION_BLOCK

// Given an X, find which of 3 tables to look in
FUNCTION fctGetTableNumberT3
  // Return a 1, 2, or 3 for which table to look in
  // NOTE: X values in each table need to be sorted in ascending order
  // NOTE: It is assumed that x values in table 1 < table 2 < table 3

  // If value is less than or equal the last value in table 1,
  // then the value must represented in or before table 1. Return 1.
  IF xVal <= t1.xVals[t1.numberOfVals - 1] THEN
    fctGetTableNumberT3 := 1;
    RETURN;
  ELSIF xVal >= t3.xVals[0] THEN
    // If value is greater than or equal to the first value in table 3,
    // then the value must be represented in or after table 3. Return 3.
    fctGetTableNumberT3 := 3;
    RETURN;
  ELSE
    // The value must be too big to be represented in table 1,
    // and too small to be represented in table 3.
    // Table 2 is the best choice. Return 2.
    fctGetTableNumberT3 := 2;
    RETURN;
  END_IF;

END_FUNCTION

// Given a table, swap the X and Y values
FUNCTION fctSwapTableT3
  // Make sure number of values does not overrun the array sizes
  length := MIN(SIZEOF(tVals) / SIZEOF(tVals[0]), SIZEOF(table.xVals) / SIZEOF(table.xVals[0]), SIZEOF(table.yVals) / SIZEOF(table.yVals[0]));
  // Y -> temp
  // X -> Y
  // temp -> X
  // nextAddr := brsmemcpy(ADR(Dest),ADR(Src),length);
  nextAddr := brsmemcpy(ADR(tVals), ADR(table.yVals), length);
  nextAddr := brsmemcpy(ADR(table.yVals), ADR(table.xVals), length);
  nextAddr := brsmemcpy(ADR(table.xVals), ADR(tVals), length);
END_FUNCTION
```

- Visualisation Logical/mappView (not shown)

### Package Logical/Libraries - Global libraries

### Library Logical/Libraries/GAProcIO (Iec) - Scale Analog functions

#### GAProcIO.typ - Exported data types
```iecst
(********************************************************************
 * COPYRIGHT -- General Atomics
 ********************************************************************
 * Library: GAProcIO
 * File: GAProcIO.typ
 * Author: Administrator
 * Created: September 11, 2015
 ********************************************************************
 * Data types of library GAProcIO
 ********************************************************************)

TYPE
	eGAPIO_RAW_SCALE_TYPE :
		(
		GAPIO_RWST_OFF := 0, (* do not process the chanel *)
		GAPIO_RWST_USINT := 1,
		GAPIO_RWST_SINT := 2,
		GAPIO_RWST_UINT := 3,
		GAPIO_RWST_INT := 4,
		GAPIO_RWST_UDINT := 5,
		GAPIO_RWST_DINT := 6,
    GAPIO_RWST_REAL := 7 (* LREAL not suppoeted by scaling routine *)
    (* RWST_LREAL := 8 *)
  ) := GAPIO_RWST_INT; (* default to int, since this is what most AIs are *)

  eGAPIO_PB_BEHAVIOR_TYPE :
    (
    GAPIO_PBBT_DISABLED   := 0, (* always off *)
    GAPIO_PBBT_MOMENTARY  := 1, (* active while pressed *)
    GAPIO_PBBT_OS_ON      := 2, (* oneshot on. Needs rising edge to turn on for 1 scan *)
    GAPIO_PBBT_PRESS_ON   := 3, (* press to turn on *)
    GAPIO_PBBT_PULSE_ON   := 4, (* turn on for a pulse *)
    GAPIO_PBBT_PRESS_OFF  := 5, (* press to turn off *)
    GAPIO_PBBT_TOGGLE     := 6  (* press to toggle *)
  ) := GAPIO_PBBT_MOMENTARY;

  sAnalogInput : 	STRUCT  (* 32 byte structure *)
    ModuleOk : BOOL; (* byte 0 H=okay *)
    ChannelOk : BOOL; (* byte 1 H=okay *)
    InRawUSINT : USINT; (* byte 2 *)
    InRawSINT : SINT; (* byte 3 *)
    InRawUINT : UINT; (* bytes 4-5 *)
    InRawINT : INT; (* bytes 6-7 *)
    InRawUDINT : UDINT; (* bytes 8-11 *)
    InRawDINT : DINT; (* bytes 12-15 *)
    InRawREAL : REAL; (* bytes 16-19 *)
    InScaled : REAL; (* byte 20-23 *)
    InScaledFiltered : REAL; (* byte 24-27 *)
    (* alarms *)
    (* bit packed integer - used so non-zero value means at least one alarm is active *)
    alms : UDINT := 0; (* b0:LoRange,b1:HiRange,b2:LoLoAlm,b3:LoAlm,b4:HiAlm,b5:HiHiAlm,b31:chErr *)
  END_STRUCT;

	sAnalogInputParams : 	STRUCT  (* analog scaling and alarm parameters *) (* raw scale type - how to interpret InRawBuffer *)
		LpEnable : BOOL := FALSE; (* turn off Low Pass Filter by default *)
		LpPreserveUnfiltered : BOOL := TRUE; (* F: unfiltered = filtered, T: keep separate *)
		AlmEnable : BOOL := FALSE;
		AlmLoLoEnable : BOOL := FALSE;
		AlmLoEnable : BOOL := FALSE;
		AlmHiEnable : BOOL := FALSE;
		AlmHiHiEnable : BOOL := FALSE; (* alarm thresholds - compare to EU (scaled) values *) (* disable range check and alarm thresholds by default if not specified *)
		RawType : eGAPIO_RAW_SCALE_TYPE := GAPIO_RWST_INT; (* default to int, since this is what most AIs are *) (* scaling parameters *)
		RawMin : REAL := 0.0; (* scale to 15 bits if not specified - a common value for ai modules *)
		RawMax : REAL := 32767.0;
		EuMin : REAL := 0.0; (* scale to percent if not specified *)
		EuMax : REAL := 100.0;
		RawOffset : REAL := 0.0; (* +/- counts value added to the raw value before scaling *)
		EuOffset : REAL := 0.0; (* +/- EU value added to EU after scaling *) (* Low Pass (Noise) filter parameters *)
		LpCoeff : REAL := 0.0; (* >=0 and <1. 0= no filtering. 0.99999= heavy filtering. *) (* alarm enables *) (* turn on or off all alarming except for out of range alarms *)
		AlmRangeThreshLo : REAL := -1.0E9;
		AlmRangeThreshHi : REAL := 1.0E9;
		AlmThreshLoLo : REAL := -1.0E9;
		AlmThreshLo : REAL := -1.0E9;
		AlmThreshHi : REAL := 1.0E9;
		AlmThreshHiHi : REAL := 1.0E9; (* alarm deadbands *) (* in % of range EU range *) (* use 0 to disable *)
		AlmDbLoPct : REAL := 1.0; (* pvs must rise above threshold by the corresponding value in order to be considered clear *)
		AlmDbHiPct : REAL := 1.0; (* pvs must drop below threshold by the corresponding value in order to be considered clear *) (* alarm time delays *) (* use 0 time to disable *)
		AlmLoOnDlyTime : TIME := T#1s;
		AlmHiOnDlyTime : TIME := T#1s; (* alarm off delay time - condition must clear for this long before being considered "gone" *)
		AlmLoOffDlyTime : TIME := T#1s;
		AlmHiOffDlyTime : TIME := T#1s;
  END_STRUCT;

  sDigitalInput : 	STRUCT
    ModuleOk : BOOL; (* H=okay *)
    ChannelOk : BOOL; (* H=okay *)
    InRaw : BOOL; (* raw input signal *)
    Value : BOOL; (* conditioned value *)
    spareBytes5_7 : ARRAY[5..7]OF BYTE;
    (* alarms *)
    (* bit packed integer - used so non-zero value means at least one alarm is active *)
    alms : UDINT := 0; (* b3:LoAlm,b4:HiAlm,b31:ch err,b0-2:reserved,b5-30:reserved *)
  END_STRUCT;

  sDigitalInputParams : 	STRUCT  (* digital signal processing and alarm parameters *)
    Enable : BOOL; (* H=process *)
    AlmEnable : BOOL := FALSE; (* set to process alarm *)
		AlmLoEnable : BOOL := FALSE; (* set to enable alarm if value is low *)
		AlmHiEnable : BOOL := FALSE; (* set to enable alarm if value is high *)
		Invert : BOOL := FALSE;
		OnDlyTime : TIME := T#0ms; (* delay time for value turning on *)
		OffDlyTime : TIME := T#0ms; (* delay time for value turning off *)
		AlmLoOnDlyTime : TIME := T#1s;
		AlmHiOnDlyTime : TIME := T#1s;
		AlmLoOffDlyTime : TIME := T#1s;
		AlmHiOffDlyTime : TIME := T#1s;
  END_STRUCT;

END_TYPE
```
